LIN {X 0,Y 361.858,Z 207.02,A -85,B 0,C 180,E1 -12997.223,E2 -12997.223} C_VEL
LIN {X 0,Y 361.83,Z 207.034,A -85,B 0,C 180,E1 -13000.756,E2 -13000.756} C_VEL
LIN {X 0,Y 361.812,Z 207.04,A -85,B 0,C 180,E1 -13004.369,E2 -13004.369} C_VEL
LIN {X 0,Y 361.828,Z 207.039,A -85,B 0,C 180,E1 -13007.569,E2 -13007.569} C_VEL
LIN {X 0,Y 361.879,Z 207.126,A -85,B 0,C 180,E1 -13011.447,E2 -13011.447} C_VEL
LIN {X 0,Y 365.809,Z 219.947,A -85,B 0,C 180,E1 -13014.488,E2 -13014.488} C_VEL
LIN {X 0,Y 369.445,Z 233.39,A -85,B 0,C 180,E1 -13017.402,E2 -13017.402} C_VEL
LIN {X 0,Y 372.235,Z 244.85,A -85,B 0,C 180,E1 -13019.72,E2 -13019.72} C_VEL
LIN {X 0,Y 373.066,Z 248.951,A -85,B 0,C 180,E1 -13019.921,E2 -13019.921} C_VEL
LIN {X 0,Y 377.476,Z 275.58,A -85,B 0,C 180,E1 -13020.87,E2 -13020.87} C_VEL
LIN {X 0,Y 378.031,Z 280.109,A -85,B 0,C 180,E1 -13021.013,E2 -13021.013} C_VEL
LIN {X 0,Y 374.715,Z 405.34,A -85,B 0,C 180,E1 -13023.549,E2 -13023.549} C_VEL
LIN {X 0,Y 373.825,Z 420.56,A -85,B 0,C 180,E1 -13024.044,E2 -13024.044} C_VEL
LIN {X 0,Y 372.576,Z 436.071,A -85,B 0,C 180,E1 -13024.78,E2 -13024.78} C_VEL
LIN {X 0,Y 371.215,Z 450.264,A -85,B 0,C 180,E1 -13025.684,E2 -13025.684} C_VEL
LIN {X 0,Y 369.635,Z 463.713,A -85,B 0,C 180,E1 -13026.764,E2 -13026.764} C_VEL
LIN {X 0,Y 367.883,Z 477.375,A -85,B 0,C 180,E1 -13028.129,E2 -13028.129} C_VEL
LIN {X 0,Y 366.23,Z 489.771,A -85,B 0,C 180,E1 -13029.647,E2 -13029.647} C_VEL
LIN {X 0,Y 364.935,Z 500.221,A -85,B 0,C 180,E1 -13031.182,E2 -13031.182} C_VEL
LIN {X 0,Y 363.602,Z 509.844,A -85,B 0,C 180,E1 -13032.857,E2 -13032.857} C_VEL
LIN {X 0,Y 362.442,Z 519.299,A -85,B 0,C 180,E1 -13034.825,E2 -13034.825} C_VEL
LIN {X 0,Y 361.565,Z 527.133,A -85,B 0,C 180,E1 -13036.798,E2 -13036.798} C_VEL
LIN {X 0,Y 360.999,Z 533.592,A -85,B 0,C 180,E1 -13038.774,E2 -13038.774} C_VEL
LIN {X 0,Y 360.557,Z 539.494,A -85,B 0,C 180,E1 -13041.029,E2 -13041.029} C_VEL
LIN {X 0,Y 360.387,Z 543.966,A -85,B 0,C 180,E1 -13043.281,E2 -13043.281} C_VEL
LIN {X 0,Y 360.351,Z 547.107,A -85,B 0,C 180,E1 -13045.526,E2 -13045.526} C_VEL
LIN {X 0,Y 360.384,Z 548.979,A -85,B 0,C 180,E1 -13047.765,E2 -13047.765} C_VEL
LIN {X 0,Y 360.474,Z 549.615,A -85,B 0,C 180,E1 -13050,E2 -13050} C_VEL
LIN {X 0,Y 360.384,Z 548.971,A -85,B 0,C 180,E1 -13052.236,E2 -13052.236} C_VEL
LIN {X 0,Y 360.384,Z 547.091,A -85,B 0,C 180,E1 -13054.474,E2 -13054.474} C_VEL
LIN {X 0,Y 360.477,Z 543.95,A -85,B 0,C 180,E1 -13056.718,E2 -13056.718} C_VEL
LIN {X 0,Y 360.559,Z 539.471,A -85,B 0,C 180,E1 -13058.971,E2 -13058.971} C_VEL
LIN {X 0,Y 361.002,Z 533.555,A -85,B 0,C 180,E1 -13061.226,E2 -13061.226} C_VEL
LIN {X 0,Y 361.685,Z 526.041,A -85,B 0,C 180,E1 -13063.484,E2 -13063.484} C_VEL
LIN {X 0,Y 362.613,Z 517.975,A -85,B 0,C 180,E1 -13065.456,E2 -13065.456} C_VEL
LIN {X 0,Y 363.789,Z 508.252,A -85,B 0,C 180,E1 -13067.424,E2 -13067.424} C_VEL
LIN {X 0,Y 365.118,Z 498.314,A -85,B 0,C 180,E1 -13069.101,E2 -13069.101} C_VEL
LIN {X 0,Y 366.636,Z 486.473,A -85,B 0,C 180,E1 -13070.771,E2 -13070.771} C_VEL
LIN {X 0,Y 368.201,Z 474.69,A -85,B 0,C 180,E1 -13072.147,E2 -13072.147} C_VEL
LIN {X 0,Y 369.832,Z 461.965,A -85,B 0,C 180,E1 -13073.372,E2 -13073.372} C_VEL
LIN {X 0,Y 371.43,Z 448.089,A -85,B 0,C 180,E1 -13074.451,E2 -13074.451} C_VEL
LIN {X 0,Y 372.66,Z 434.821,A -85,B 0,C 180,E1 -13075.275,E2 -13075.275} C_VEL
LIN {X 0,Y 373.81,Z 420.208,A -85,B 0,C 180,E1 -13075.958,E2 -13075.958} C_VEL
LIN {X 0,Y 374.684,Z 404.745,A -85,B 0,C 180,E1 -13076.454,E2 -13076.454} C_VEL
LIN {X 0,Y 377.559,Z 296.462,A -85,B 0,C 180,E1 -13078.649,E2 -13078.649} C_VEL
LIN {X 0,Y 377.872,Z 278.457,A -85,B 0,C 180,E1 -13079.019,E2 -13079.019} C_VEL
LIN {X 0,Y 372.834,Z 247.587,A -85,B 0,C 180,E1 -13080.112,E2 -13080.112} C_VEL
LIN {X 0,Y 372.193,Z 244.833,A -85,B 0,C 180,E1 -13080.272,E2 -13080.272} C_VEL
LIN {X 0,Y 369.443,Z 233.326,A -85,B 0,C 180,E1 -13082.6,E2 -13082.6} C_VEL
LIN {X 0,Y 365.814,Z 219.862,A -85,B 0,C 180,E1 -13085.517,E2 -13085.517} C_VEL
LIN {X 0,Y 361.901,Z 207.157,A -85,B 0,C 180,E1 -13088.533,E2 -13088.533} C_VEL
LIN {X 0,Y 361.82,Z 207.013,A -85,B 0,C 180,E1 -13091.331,E2 -13091.331} C_VEL
LIN {X 0,Y 361.815,Z 207.03,A -85,B 0,C 180,E1 -13094.369,E2 -13094.369} C_VEL
LIN {X 0,Y 361.834,Z 207.026,A -85,B 0,C 180,E1 -13097.568,E2 -13097.568} C_VEL
LIN {X 0,Y 361.868,Z 207.03,A -85,B 0,C 180,E1 -13100.973,E2 -13100.973} C_VEL
LIN {X 0,Y 361.872,Z 207.038,A -85,B 0,C 180,E1 -13104.655,E2 -13104.655} C_VEL
LIN {X 0,Y 361.835,Z 207.02,A -85,B 0,C 180,E1 -13108.371,E2 -13108.371} C_VEL
LIN {X 0,Y 361.899,Z 207.028,A -85,B 0,C 180,E1 -13110.955,E2 -13110.955} C_VEL
LIN {X 0,Y 361.952,Z 206.995,A -85,B 0,C 180,E1 -13113.475,E2 -13113.475} C_VEL
LIN {X 0,Y 361.888,Z 207.03,A -85,B 0,C 180,E1 -13117.145,E2 -13117.145} C_VEL
LIN {X 0,Y 361.919,Z 207.026,A -85,B 0,C 180,E1 -13120.724,E2 -13120.724} C_VEL
LIN {X 0,Y 361.944,Z 207.026,A -85,B 0,C 180,E1 -13124.226,E2 -13124.226} C_VEL
LIN {X 0,Y 361.997,Z 207.012,A -85,B 0,C 180,E1 -13126.528,E2 -13126.528} C_VEL
LIN {X 0,Y 362.029,Z 207.007,A -85,B 0,C 180,E1 -13129.938,E2 -13129.938} C_VEL
LIN {X 0,Y 362.161,Z 206.997,A -85,B 0,C 180,E1 -13133.314,E2 -13133.314} C_VEL
LIN {X 0,Y 362.278,Z 206.978,A -85,B 0,C 180,E1 -13137.777,E2 -13137.777} C_VEL
LIN {X 0,Y 362.424,Z 206.963,A -85,B 0,C 180,E1 -13140,E2 -13140} C_VEL
LIN {X 0,Y 362.278,Z 206.977,A -85,B 0,C 180,E1 -13142.224,E2 -13142.224} C_VEL
LIN {X 0,Y 362.17,Z 206.993,A -85,B 0,C 180,E1 -13146.686,E2 -13146.686} C_VEL
LIN {X 0,Y 362.073,Z 207.005,A -85,B 0,C 180,E1 -13148.933,E2 -13148.933} C_VEL
LIN {X 0,Y 361.958,Z 207.015,A -85,B 0,C 180,E1 -13152.333,E2 -13152.333} C_VEL
LIN {X 0,Y 361.961,Z 207.022,A -85,B 0,C 180,E1 -13154.621,E2 -13154.621} C_VEL
LIN {X 0,Y 361.955,Z 207.022,A -85,B 0,C 180,E1 -13158.1,E2 -13158.1} C_VEL
LIN {X 0,Y 361.892,Z 207.031,A -85,B 0,C 180,E1 -13161.653,E2 -13161.653} C_VEL
LIN {X 0,Y 361.927,Z 207.029,A -85,B 0,C 180,E1 -13165.29,E2 -13165.29} C_VEL
LIN {X 0,Y 361.907,Z 207.01,A -85,B 0,C 180,E1 -13167.779,E2 -13167.779} C_VEL
LIN {X 0,Y 361.837,Z 207.038,A -85,B 0,C 180,E1 -13171.63,E2 -13171.63} C_VEL
LIN {X 0,Y 361.874,Z 207.015,A -85,B 0,C 180,E1 -13175.345,E2 -13175.345} C_VEL
LIN {X 0,Y 361.869,Z 207.02,A -85,B 0,C 180,E1 -13179.027,E2 -13179.027} C_VEL
LIN {X 0,Y 361.836,Z 207.035,A -85,B 0,C 180,E1 -13182.829,E2 -13182.829} C_VEL
LIN {X 0,Y 361.819,Z 207.041,A -85,B 0,C 180,E1 -13185.947,E2 -13185.947} C_VEL
LIN {X 0,Y 361.837,Z 207.04,A -85,B 0,C 180,E1 -13189.245,E2 -13189.245} C_VEL
LIN {X 0,Y 361.872,Z 207.03,A -85,B 0,C 180,E1 -13192.776,E2 -13192.776} C_VEL
LIN {X 0,Y 361.897,Z 207.231,A -85,B 0,C 180,E1 -13193.593,E2 -13193.593} C_VEL
LIN {X 0,Y 364.857,Z 217.605,A -85,B 0,C 180,E1 -13196.315,E2 -13196.315} C_VEL
LIN {X 0,Y 367.533,Z 228.193,A -85,B 0,C 180,E1 -13198.916,E2 -13198.916} C_VEL
LIN {X 0,Y 370.249,Z 240.049,A -85,B 0,C 180,E1 -13201.67,E2 -13201.67} C_VEL
LIN {X 0,Y 370.322,Z 243.02,A -85,B 0,C 180,E1 -13202.292,E2 -13202.292} C_VEL
LIN {X 0,Y 370.224,Z 244.579,A -85,B 0,C 180,E1 -13202.552,E2 -13202.552} C_VEL
LIN {X 0,Y 376.066,Z 272.726,A -85,B 0,C 180,E1 -13203.636,E2 -13203.636} C_VEL
LIN {X 0,Y 377.412,Z 280.727,A -85,B 0,C 180,E1 -13203.904,E2 -13203.904} C_VEL
LIN {X 0,Y 375.224,Z 388.776,A -85,B 0,C 180,E1 -13205.886,E2 -13205.886} C_VEL
LIN {X 0,Y 374.523,Z 402.901,A -85,B 0,C 180,E1 -13206.353,E2 -13206.353} C_VEL
LIN {X 0,Y 373.655,Z 416.248,A -85,B 0,C 180,E1 -13207.005,E2 -13207.005} C_VEL
LIN {X 0,Y 372.396,Z 429.002,A -85,B 0,C 180,E1 -13207.824,E2 -13207.824} C_VEL
LIN {X 0,Y 371.049,Z 441.949,A -85,B 0,C 180,E1 -13208.907,E2 -13208.907} C_VEL
LIN {X 0,Y 369.441,Z 453.698,A -85,B 0,C 180,E1 -13210.12,E2 -13210.12} C_VEL
LIN {X 0,Y 368.1,Z 463.475,A -85,B 0,C 180,E1 -13211.349,E2 -13211.349} C_VEL
LIN {X 0,Y 366.399,Z 474.26,A -85,B 0,C 180,E1 -13212.991,E2 -13212.991} C_VEL
LIN {X 0,Y 365.128,Z 483.181,A -85,B 0,C 180,E1 -13214.653,E2 -13214.653} C_VEL
LIN {X 0,Y 363.659,Z 491.735,A -85,B 0,C 180,E1 -13216.59,E2 -13216.59} C_VEL
LIN {X 0,Y 362.727,Z 497.801,A -85,B 0,C 180,E1 -13218.261,E2 -13218.261} C_VEL
LIN {X 0,Y 361.781,Z 504.251,A -85,B 0,C 180,E1 -13220.495,E2 -13220.495} C_VEL
LIN {X 0,Y 361.304,Z 508.07,A -85,B 0,C 180,E1 -13222.174,E2 -13222.174} C_VEL
LIN {X 0,Y 360.869,Z 511.89,A -85,B 0,C 180,E1 -13224.412,E2 -13224.412} C_VEL
LIN {X 0,Y 360.604,Z 514.38,A -85,B 0,C 180,E1 -13226.648,E2 -13226.648} C_VEL
LIN {X 0,Y 360.499,Z 515.621,A -85,B 0,C 180,E1 -13228.883,E2 -13228.883} C_VEL
LIN {X 0,Y 360.497,Z 515.649,A -85,B 0,C 180,E1 -13231.117,E2 -13231.117} C_VEL
LIN {X 0,Y 360.594,Z 514.467,A -85,B 0,C 180,E1 -13233.352,E2 -13233.352} C_VEL
LIN {X 0,Y 360.857,Z 512.038,A -85,B 0,C 180,E1 -13235.588,E2 -13235.588} C_VEL
LIN {X 0,Y 361.286,Z 508.284,A -85,B 0,C 180,E1 -13237.826,E2 -13237.826} C_VEL
LIN {X 0,Y 361.943,Z 503.077,A -85,B 0,C 180,E1 -13240.064,E2 -13240.064} C_VEL
LIN {X 0,Y 362.965,Z 496.242,A -85,B 0,C 180,E1 -13242.297,E2 -13242.297} C_VEL
LIN {X 0,Y 364.222,Z 488.716,A -85,B 0,C 180,E1 -13244.242,E2 -13244.242} C_VEL
LIN {X 0,Y 365.555,Z 479.746,A -85,B 0,C 180,E1 -13246.129,E2 -13246.129} C_VEL
LIN {X 0,Y 366.277,Z 475.133,A -85,B 0,C 180,E1 -13246.961,E2 -13246.961} C_VEL
LIN {X 0,Y 366.252,Z 471.21,A -85,B 0,C 180,E1 -13247.651,E2 -13247.651} C_VEL
LIN {X 0,Y 364.53,Z 464.68,A -85,B 0,C 180,E1 -13248.791,E2 -13248.791} C_VEL
LIN {X 0,Y 362.904,Z 457.796,A -85,B 0,C 180,E1 -13249.881,E2 -13249.881} C_VEL
LIN {X 0,Y 362.989,Z 453.195,A -85,B 0,C 180,E1 -13250.469,E2 -13250.469} C_VEL
LIN {X 0,Y 364.736,Z 440.566,A -85,B 0,C 180,E1 -13251.772,E2 -13251.772} C_VEL
LIN {X 0,Y 366.108,Z 427.91,A -85,B 0,C 180,E1 -13252.814,E2 -13252.814} C_VEL
LIN {X 0,Y 367.367,Z 414.082,A -85,B 0,C 180,E1 -13253.687,E2 -13253.687} C_VEL
LIN {X 0,Y 368.307,Z 400.048,A -85,B 0,C 180,E1 -13254.333,E2 -13254.333} C_VEL
LIN {X 0,Y 368.949,Z 385.269,A -85,B 0,C 180,E1 -13254.775,E2 -13254.775} C_VEL
LIN {X 0,Y 371.083,Z 280.253,A -85,B 0,C 180,E1 -13256.723,E2 -13256.723} C_VEL
LIN {X 0,Y 364.68,Z 248.87,A -85,B 0,C 180,E1 -13257.924,E2 -13257.924} C_VEL
LIN {X 0,Y 363.707,Z 244.456,A -85,B 0,C 180,E1 -13258.139,E2 -13258.139} C_VEL
LIN {X 0,Y 363.246,Z 240.748,A -85,B 0,C 180,E1 -13258.926,E2 -13258.926} C_VEL
LIN {X 0,Y 360.536,Z 228.921,A -85,B 0,C 180,E1 -13261.756,E2 -13261.756} C_VEL
LIN {X 0,Y 357.479,Z 217.065,A -85,B 0,C 180,E1 -13264.759,E2 -13264.759} C_VEL
LIN {X 0,Y 354.825,Z 207.985,A -85,B 0,C 180,E1 -13267.271,E2 -13267.271} C_VEL
LIN {X 0,Y 354.786,Z 207.92,A -85,B 0,C 180,E1 -13270.82,E2 -13270.82} C_VEL
LIN {X 0,Y 354.761,Z 207.919,A -85,B 0,C 180,E1 -13274.506,E2 -13274.506} C_VEL
LIN {X 0,Y 354.791,Z 207.918,A -85,B 0,C 180,E1 -13277.662,E2 -13277.662} C_VEL
LIN {X 0,Y 354.811,Z 207.897,A -85,B 0,C 180,E1 -13280.665,E2 -13280.665} C_VEL
LIN {X 0,Y 354.818,Z 207.899,A -85,B 0,C 180,E1 -13284.3,E2 -13284.3} C_VEL
LIN {X 0,Y 354.785,Z 207.918,A -85,B 0,C 180,E1 -13287.666,E2 -13287.666} C_VEL
LIN {X 0,Y 354.864,Z 207.882,A -85,B 0,C 180,E1 -13290.621,E2 -13290.621} C_VEL
LIN {X 0,Y 354.894,Z 207.901,A -85,B 0,C 180,E1 -13294.172,E2 -13294.172} C_VEL
LIN {X 0,Y 354.829,Z 207.91,A -85,B 0,C 180,E1 -13297.893,E2 -13297.893} C_VEL
LIN {X 0,Y 354.917,Z 207.899,A -85,B 0,C 180,E1 -13301.891,E2 -13301.891} C_VEL
LIN {X 0,Y 354.936,Z 207.897,A -85,B 0,C 180,E1 -13305.981,E2 -13305.981} C_VEL
LIN {X 0,Y 354.971,Z 207.891,A -85,B 0,C 180,E1 -13309.735,E2 -13309.735} C_VEL
LIN {X 0,Y 355.107,Z 207.869,A -85,B 0,C 180,E1 -13312.037,E2 -13312.037} C_VEL
LIN {X 0,Y 355.086,Z 207.879,A -85,B 0,C 180,E1 -13314.32,E2 -13314.32} C_VEL
LIN {X 0,Y 355.239,Z 207.853,A -85,B 0,C 180,E1 -13317.732,E2 -13317.732} C_VEL
LIN {X 0,Y 355.391,Z 207.839,A -85,B 0,C 180,E1 -13320,E2 -13320} C_VEL
LIN {X 0,Y 355.239,Z 207.854,A -85,B 0,C 180,E1 -13322.267,E2 -13322.267} C_VEL
LIN {X 0,Y 355.131,Z 207.873,A -85,B 0,C 180,E1 -13326.819,E2 -13326.819} C_VEL
LIN {X 0,Y 355.008,Z 207.882,A -85,B 0,C 180,E1 -13329.112,E2 -13329.112} C_VEL
LIN {X 0,Y 354.914,Z 207.897,A -85,B 0,C 180,E1 -13332.581,E2 -13332.581} C_VEL
LIN {X 0,Y 354.883,Z 207.905,A -85,B 0,C 180,E1 -13336.096,E2 -13336.096} C_VEL
LIN {X 0,Y 354.9,Z 207.898,A -85,B 0,C 180,E1 -13338.472,E2 -13338.472} C_VEL
LIN {X 0,Y 354.828,Z 207.907,A -85,B 0,C 180,E1 -13342.106,E2 -13342.106} C_VEL
LIN {X 0,Y 354.893,Z 207.877,A -85,B 0,C 180,E1 -13345.828,E2 -13345.828} C_VEL
LIN {X 0,Y 354.848,Z 207.912,A -85,B 0,C 180,E1 -13349.679,E2 -13349.679} C_VEL
LIN {X 0,Y 354.8,Z 207.899,A -85,B 0,C 180,E1 -13353.702,E2 -13353.702} C_VEL
LIN {X 0,Y 354.792,Z 207.907,A -85,B 0,C 180,E1 -13356.46,E2 -13356.46} C_VEL
LIN {X 0,Y 354.819,Z 207.912,A -85,B 0,C 180,E1 -13359.424,E2 -13359.424} C_VEL
LIN {X 0,Y 354.783,Z 207.908,A -85,B 0,C 180,E1 -13362.868,E2 -13362.868} C_VEL
LIN {X 0,Y 354.761,Z 207.91,A -85,B 0,C 180,E1 -13366.104,E2 -13366.104} C_VEL
LIN {X 0,Y 354.777,Z 207.88,A -85,B 0,C 180,E1 -13369.179,E2 -13369.179} C_VEL
LIN {X 0,Y 354.846,Z 208.08,A -85,B 0,C 180,E1 -13370.784,E2 -13370.784} C_VEL
LIN {X 0,Y 358.939,Z 221.433,A -85,B 0,C 180,E1 -13374.029,E2 -13374.029} C_VEL
LIN {X 0,Y 362.471,Z 234.285,A -85,B 0,C 180,E1 -13376.904,E2 -13376.904} C_VEL
LIN {X 0,Y 365.188,Z 245.142,A -85,B 0,C 180,E1 -13379.137,E2 -13379.137} C_VEL
LIN {X 0,Y 366.628,Z 248.786,A -85,B 0,C 180,E1 -13379.367,E2 -13379.367} C_VEL
LIN {X 0,Y 370.877,Z 274.547,A -85,B 0,C 180,E1 -13380.311,E2 -13380.311} C_VEL
LIN {X 0,Y 371.729,Z 281.26,A -85,B 0,C 180,E1 -13380.531,E2 -13380.531} C_VEL
LIN {X 0,Y 368.294,Z 405.657,A -85,B 0,C 180,E1 -13383.089,E2 -13383.089} C_VEL
LIN {X 0,Y 367.319,Z 421.492,A -85,B 0,C 180,E1 -13383.626,E2 -13383.626} C_VEL
LIN {X 0,Y 366.057,Z 436.211,A -85,B 0,C 180,E1 -13384.345,E2 -13384.345} C_VEL
LIN {X 0,Y 364.716,Z 449.758,A -85,B 0,C 180,E1 -13385.222,E2 -13385.222} C_VEL
LIN {X 0,Y 363.065,Z 463.252,A -85,B 0,C 180,E1 -13386.318,E2 -13386.318} C_VEL
LIN {X 0,Y 361.254,Z 476.962,A -85,B 0,C 180,E1 -13387.707,E2 -13387.707} C_VEL
LIN {X 0,Y 359.509,Z 489.38,A -85,B 0,C 180,E1 -13389.249,E2 -13389.249} C_VEL
LIN {X 0,Y 358.111,Z 499.836,A -85,B 0,C 180,E1 -13390.81,E2 -13390.81} C_VEL
LIN {X 0,Y 356.744,Z 509.473,A -85,B 0,C 180,E1 -13392.517,E2 -13392.517} C_VEL
LIN {X 0,Y 355.511,Z 518.939,A -85,B 0,C 180,E1 -13394.522,E2 -13394.522} C_VEL
LIN {X 0,Y 354.555,Z 526.779,A -85,B 0,C 180,E1 -13396.532,E2 -13396.532} C_VEL
LIN {X 0,Y 353.952,Z 533.245,A -85,B 0,C 180,E1 -13398.548,E2 -13398.548} C_VEL
LIN {X 0,Y 353.498,Z 539.153,A -85,B 0,C 180,E1 -13400.849,E2 -13400.849} C_VEL
LIN {X 0,Y 353.305,Z 543.629,A -85,B 0,C 180,E1 -13403.146,E2 -13403.146} C_VEL
LIN {X 0,Y 353.262,Z 546.772,A -85,B 0,C 180,E1 -13405.436,E2 -13405.436} C_VEL
LIN {X 0,Y 353.285,Z 548.646,A -85,B 0,C 180,E1 -13407.72,E2 -13407.72} C_VEL
LIN {X 0,Y 353.393,Z 549.283,A -85,B 0,C 180,E1 -13410,E2 -13410} C_VEL
LIN {X 0,Y 353.285,Z 548.638,A -85,B 0,C 180,E1 -13412.281,E2 -13412.281} C_VEL
LIN {X 0,Y 353.295,Z 546.756,A -85,B 0,C 180,E1 -13414.564,E2 -13414.564} C_VEL
LIN {X 0,Y 353.383,Z 543.611,A -85,B 0,C 180,E1 -13416.854,E2 -13416.854} C_VEL
LIN {X 0,Y 353.499,Z 539.128,A -85,B 0,C 180,E1 -13419.152,E2 -13419.152} C_VEL
LIN {X 0,Y 353.957,Z 533.206,A -85,B 0,C 180,E1 -13421.453,E2 -13421.453} C_VEL
LIN {X 0,Y 354.72,Z 525.687,A -85,B 0,C 180,E1 -13423.754,E2 -13423.754} C_VEL
LIN {X 0,Y 355.674,Z 517.61,A -85,B 0,C 180,E1 -13425.765,E2 -13425.765} C_VEL
LIN {X 0,Y 356.957,Z 507.879,A -85,B 0,C 180,E1 -13427.769,E2 -13427.769} C_VEL
LIN {X 0,Y 358.534,Z 496.723,A -85,B 0,C 180,E1 -13429.663,E2 -13429.663} C_VEL
LIN {X 0,Y 359.929,Z 486.064,A -85,B 0,C 180,E1 -13431.176,E2 -13431.176} C_VEL
LIN {X 0,Y 361.605,Z 474.256,A -85,B 0,C 180,E1 -13432.573,E2 -13432.573} C_VEL
LIN {X 0,Y 363.245,Z 461.488,A -85,B 0,C 180,E1 -13433.821,E2 -13433.821} C_VEL
LIN {X 0,Y 364.918,Z 447.555,A -85,B 0,C 180,E1 -13434.916,E2 -13434.916} C_VEL
LIN {X 0,Y 366.277,Z 433.522,A -85,B 0,C 180,E1 -13435.787,E2 -13435.787} C_VEL
LIN {X 0,Y 367.489,Z 418.521,A -85,B 0,C 180,E1 -13436.477,E2 -13436.477} C_VEL
LIN {X 0,Y 368.325,Z 403.593,A -85,B 0,C 180,E1 -13436.947,E2 -13436.947} C_VEL
LIN {X 0,Y 371.686,Z 280.699,A -85,B 0,C 180,E1 -13439.467,E2 -13439.467} C_VEL
LIN {X 0,Y 367.099,Z 251.451,A -85,B 0,C 180,E1 -13440.514,E2 -13440.514} C_VEL
LIN {X 0,Y 366.131,Z 247.57,A -85,B 0,C 180,E1 -13440.687,E2 -13440.687} C_VEL
LIN {X 0,Y 365.05,Z 244.821,A -85,B 0,C 180,E1 -13440.891,E2 -13440.891} C_VEL
LIN {X 0,Y 362.081,Z 232.745,A -85,B 0,C 180,E1 -13443.423,E2 -13443.423} C_VEL
LIN {X 0,Y 358.606,Z 220.27,A -85,B 0,C 180,E1 -13446.224,E2 -13446.224} C_VEL
LIN {X 0,Y 354.843,Z 208.045,A -85,B 0,C 180,E1 -13449.217,E2 -13449.217} C_VEL
LIN {X 0,Y 354.785,Z 207.919,A -85,B 0,C 180,E1 -13452.867,E2 -13452.867} C_VEL
LIN {X 0,Y 354.766,Z 207.92,A -85,B 0,C 180,E1 -13456.104,E2 -13456.104} C_VEL
LIN {X 0,Y 354.786,Z 207.911,A -85,B 0,C 180,E1 -13459.179,E2 -13459.179} C_VEL
LIN {X 0,Y 354.806,Z 207.898,A -85,B 0,C 180,E1 -13462.403,E2 -13462.403} C_VEL
LIN {X 0,Y 354.81,Z 207.916,A -85,B 0,C 180,E1 -13464.941,E2 -13464.941} C_VEL
LIN {X 0,Y 354.791,Z 207.897,A -85,B 0,C 180,E1 -13468.405,E2 -13468.405} C_VEL
LIN {X 0,Y 354.849,Z 207.9,A -85,B 0,C 180,E1 -13471.619,E2 -13471.619} C_VEL
LIN {X 0,Y 354.897,Z 207.876,A -85,B 0,C 180,E1 -13474.173,E2 -13474.173} C_VEL
LIN {X 0,Y 354.833,Z 207.907,A -85,B 0,C 180,E1 -13477.894,E2 -13477.894} C_VEL
LIN {X 0,Y 354.921,Z 207.894,A -85,B 0,C 180,E1 -13481.891,E2 -13481.891} C_VEL
LIN {X 0,Y 354.941,Z 207.89,A -85,B 0,C 180,E1 -13485.981,E2 -13485.981} C_VEL
LIN {X 0,Y 354.976,Z 207.886,A -85,B 0,C 180,E1 -13489.736,E2 -13489.736} C_VEL
LIN {X 0,Y 355.124,Z 207.873,A -85,B 0,C 180,E1 -13493.181,E2 -13493.181} C_VEL
LIN {X 0,Y 355.242,Z 207.855,A -85,B 0,C 180,E1 -13497.733,E2 -13497.733} C_VEL
LIN {X 0,Y 355.373,Z 207.841,A -85,B 0,C 180,E1 -13500,E2 -13500} C_VEL
LIN {X 0,Y 355.242,Z 207.853,A -85,B 0,C 180,E1 -13502.268,E2 -13502.268} C_VEL
LIN {X 0,Y 355.136,Z 207.868,A -85,B 0,C 180,E1 -13506.819,E2 -13506.819} C_VEL
LIN {X 0,Y 355.014,Z 207.886,A -85,B 0,C 180,E1 -13509.113,E2 -13509.113} C_VEL
LIN {X 0,Y 354.919,Z 207.892,A -85,B 0,C 180,E1 -13512.581,E2 -13512.581} C_VEL
LIN {X 0,Y 354.888,Z 207.894,A -85,B 0,C 180,E1 -13516.096,E2 -13516.096} C_VEL
LIN {X 0,Y 354.9,Z 207.901,A -85,B 0,C 180,E1 -13518.472,E2 -13518.472} C_VEL
LIN {X 0,Y 354.835,Z 207.909,A -85,B 0,C 180,E1 -13522.106,E2 -13522.106} C_VEL
LIN {X 0,Y 354.898,Z 207.901,A -85,B 0,C 180,E1 -13525.828,E2 -13525.828} C_VEL
LIN {X 0,Y 354.817,Z 207.891,A -85,B 0,C 180,E1 -13529.682,E2 -13529.682} C_VEL
LIN {X 0,Y 354.814,Z 207.899,A -85,B 0,C 180,E1 -13533.684,E2 -13533.684} C_VEL
LIN {X 0,Y 354.798,Z 207.908,A -85,B 0,C 180,E1 -13536.46,E2 -13536.46} C_VEL
LIN {X 0,Y 354.824,Z 207.894,A -85,B 0,C 180,E1 -13539.424,E2 -13539.424} C_VEL
LIN {X 0,Y 354.788,Z 207.912,A -85,B 0,C 180,E1 -13542.867,E2 -13542.867} C_VEL
LIN {X 0,Y 354.768,Z 207.92,A -85,B 0,C 180,E1 -13546.104,E2 -13546.104} C_VEL
LIN {X 0,Y 354.789,Z 207.918,A -85,B 0,C 180,E1 -13549.179,E2 -13549.179} C_VEL
LIN {X 0,Y 354.849,Z 208.012,A -85,B 0,C 180,E1 -13552.883,E2 -13552.883} C_VEL
LIN {X 0,Y 358.303,Z 220.102,A -85,B 0,C 180,E1 -13556.152,E2 -13556.152} C_VEL
LIN {X 0,Y 361.062,Z 231.207,A -85,B 0,C 180,E1 -13558.921,E2 -13558.921} C_VEL
LIN {X 0,Y 363.456,Z 241.708,A -85,B 0,C 180,E1 -13561.407,E2 -13561.407} C_VEL
LIN {X 0,Y 363.677,Z 244.442,A -85,B 0,C 180,E1 -13561.966,E2 -13561.966} C_VEL
LIN {X 0,Y 369.097,Z 270.076,A -85,B 0,C 180,E1 -13563.008,E2 -13563.008} C_VEL
LIN {X 0,Y 371.088,Z 280.716,A -85,B 0,C 180,E1 -13563.393,E2 -13563.393} C_VEL
LIN {X 0,Y 368.853,Z 388.562,A -85,B 0,C 180,E1 -13565.405,E2 -13565.405} C_VEL
LIN {X 0,Y 368.114,Z 402.833,A -85,B 0,C 180,E1 -13565.878,E2 -13565.878} C_VEL
LIN {X 0,Y 367.147,Z 416.969,A -85,B 0,C 180,E1 -13566.583,E2 -13566.583} C_VEL
LIN {X 0,Y 365.866,Z 429.497,A -85,B 0,C 180,E1 -13567.407,E2 -13567.407} C_VEL
LIN {X 0,Y 364.447,Z 442.397,A -85,B 0,C 180,E1 -13568.506,E2 -13568.506} C_VEL
LIN {X 0,Y 362.78,Z 454.113,A -85,B 0,C 180,E1 -13569.74,E2 -13569.74} C_VEL
LIN {X 0,Y 361.378,Z 463.866,A -85,B 0,C 180,E1 -13570.989,E2 -13570.989} C_VEL
LIN {X 0,Y 359.604,Z 474.634,A -85,B 0,C 180,E1 -13572.66,E2 -13572.66} C_VEL
LIN {X 0,Y 358.266,Z 483.544,A -85,B 0,C 180,E1 -13574.352,E2 -13574.352} C_VEL
LIN {X 0,Y 356.764,Z 492.088,A -85,B 0,C 180,E1 -13576.326,E2 -13576.326} C_VEL
LIN {X 0,Y 355.775,Z 498.146,A -85,B 0,C 180,E1 -13578.029,E2 -13578.029} C_VEL
LIN {X 0,Y 354.784,Z 504.591,A -85,B 0,C 180,E1 -13580.306,E2 -13580.306} C_VEL
LIN {X 0,Y 354.264,Z 508.41,A -85,B 0,C 180,E1 -13582.017,E2 -13582.017} C_VEL
LIN {X 0,Y 353.825,Z 512.225,A -85,B 0,C 180,E1 -13584.3,E2 -13584.3} C_VEL
LIN {X 0,Y 353.516,Z 514.715,A -85,B 0,C 180,E1 -13586.58,E2 -13586.58} C_VEL
LIN {X 0,Y 353.421,Z 515.954,A -85,B 0,C 180,E1 -13588.86,E2 -13588.86} C_VEL
LIN {X 0,Y 353.418,Z 515.981,A -85,B 0,C 180,E1 -13591.139,E2 -13591.139} C_VEL
LIN {X 0,Y 353.505,Z 514.8,A -85,B 0,C 180,E1 -13593.419,E2 -13593.419} C_VEL
LIN {X 0,Y 353.792,Z 512.372,A -85,B 0,C 180,E1 -13595.7,E2 -13595.7} C_VEL
LIN {X 0,Y 354.241,Z 508.621,A -85,B 0,C 180,E1 -13597.982,E2 -13597.982} C_VEL
LIN {X 0,Y 354.94,Z 503.419,A -85,B 0,C 180,E1 -13600.265,E2 -13600.265} C_VEL
LIN {X 0,Y 356.011,Z 496.588,A -85,B 0,C 180,E1 -13602.541,E2 -13602.541} C_VEL
LIN {X 0,Y 357.333,Z 489.07,A -85,B 0,C 180,E1 -13604.522,E2 -13604.522} C_VEL
LIN {X 0,Y 358.738,Z 480.108,A -85,B 0,C 180,E1 -13606.444,E2 -13606.444} C_VEL
LIN {X 0,Y 360.4,Z 470.14,A -85,B 0,C 180,E1 -13608.18,E2 -13608.18} C_VEL
LIN {X 0,Y 362.052,Z 459.413,A -85,B 0,C 180,E1 -13609.71,E2 -13609.71} C_VEL
LIN {X 0,Y 362.989,Z 453.195,A -85,B 0,C 180,E1 -13610.469,E2 -13610.469} C_VEL
LIN {X 0,Y 363.085,Z 448.516,A -85,B 0,C 180,E1 -13611.04,E2 -13611.04} C_VEL
LIN {X 0,Y 361.455,Z 440.814,A -85,B 0,C 180,E1 -13611.999,E2 -13611.999} C_VEL
LIN {X 0,Y 359.744,Z 432.759,A -85,B 0,C 180,E1 -13612.877,E2 -13612.877} C_VEL
LIN {X 0,Y 359.693,Z 427.53,A -85,B 0,C 180,E1 -13613.313,E2 -13613.313} C_VEL
LIN {X 0,Y 360.913,Z 414.689,A -85,B 0,C 180,E1 -13614.137,E2 -13614.137} C_VEL
LIN {X 0,Y 361.898,Z 400.827,A -85,B 0,C 180,E1 -13614.793,E2 -13614.793} C_VEL
LIN {X 0,Y 362.568,Z 386.46,A -85,B 0,C 180,E1 -13615.241,E2 -13615.241} C_VEL
LIN {X 0,Y 364.801,Z 281.372,A -85,B 0,C 180,E1 -13617.228,E2 -13617.228} C_VEL
LIN {X 0,Y 359.474,Z 254.909,A -85,B 0,C 180,E1 -13618.261,E2 -13618.261} C_VEL
LIN {X 0,Y 357.173,Z 245.429,A -85,B 0,C 180,E1 -13618.685,E2 -13618.685} C_VEL
LIN {X 0,Y 356.807,Z 244.075,A -85,B 0,C 180,E1 -13618.828,E2 -13618.828} C_VEL
LIN {X 0,Y 354.349,Z 233.053,A -85,B 0,C 180,E1 -13621.477,E2 -13621.477} C_VEL
LIN {X 0,Y 351.349,Z 221.277,A -85,B 0,C 180,E1 -13624.498,E2 -13624.498} C_VEL
LIN {X 0,Y 348.513,Z 211.254,A -85,B 0,C 180,E1 -13627.225,E2 -13627.225} C_VEL
LIN {X 0,Y 347.772,Z 208.86,A -85,B 0,C 180,E1 -13627.988,E2 -13627.988} C_VEL
LIN {X 0,Y 347.748,Z 208.783,A -85,B 0,C 180,E1 -13631.829,E2 -13631.829} C_VEL
LIN {X 0,Y 347.703,Z 208.79,A -85,B 0,C 180,E1 -13635.026,E2 -13635.026} C_VEL
LIN {X 0,Y 347.747,Z 208.795,A -85,B 0,C 180,E1 -13638.396,E2 -13638.396} C_VEL
LIN {X 0,Y 347.77,Z 208.792,A -85,B 0,C 180,E1 -13642.011,E2 -13642.011} C_VEL
LIN {X 0,Y 347.74,Z 208.773,A -85,B 0,C 180,E1 -13645.535,E2 -13645.535} C_VEL
LIN {X 0,Y 347.76,Z 208.781,A -85,B 0,C 180,E1 -13649.653,E2 -13649.653} C_VEL
LIN {X 0,Y 347.847,Z 208.764,A -85,B 0,C 180,E1 -13652.744,E2 -13652.744} C_VEL
LIN {X 0,Y 347.783,Z 208.782,A -85,B 0,C 180,E1 -13656.161,E2 -13656.161} C_VEL
LIN {X 0,Y 347.811,Z 208.776,A -85,B 0,C 180,E1 -13659.909,E2 -13659.909} C_VEL
LIN {X 0,Y 347.86,Z 208.779,A -85,B 0,C 180,E1 -13662.359,E2 -13662.359} C_VEL
LIN {X 0,Y 347.891,Z 208.774,A -85,B 0,C 180,E1 -13665.97,E2 -13665.97} C_VEL
LIN {X 0,Y 347.922,Z 208.769,A -85,B 0,C 180,E1 -13669.525,E2 -13669.525} C_VEL
LIN {X 0,Y 348.067,Z 208.747,A -85,B 0,C 180,E1 -13671.874,E2 -13671.874} C_VEL
LIN {X 0,Y 348.061,Z 208.753,A -85,B 0,C 180,E1 -13674.205,E2 -13674.205} C_VEL
LIN {X 0,Y 348.201,Z 208.73,A -85,B 0,C 180,E1 -13677.686,E2 -13677.686} C_VEL
LIN {X 0,Y 348.339,Z 208.717,A -85,B 0,C 180,E1 -13680,E2 -13680} C_VEL
LIN {X 0,Y 348.202,Z 208.731,A -85,B 0,C 180,E1 -13682.313,E2 -13682.313} C_VEL
LIN {X 0,Y 348.099,Z 208.748,A -85,B 0,C 180,E1 -13686.958,E2 -13686.958} C_VEL
LIN {X 0,Y 347.961,Z 208.76,A -85,B 0,C 180,E1 -13689.298,E2 -13689.298} C_VEL
LIN {X 0,Y 347.883,Z 208.771,A -85,B 0,C 180,E1 -13692.839,E2 -13692.839} C_VEL
LIN {X 0,Y 347.832,Z 208.78,A -85,B 0,C 180,E1 -13696.431,E2 -13696.431} C_VEL
LIN {X 0,Y 347.849,Z 208.778,A -85,B 0,C 180,E1 -13698.86,E2 -13698.86} C_VEL
LIN {X 0,Y 347.768,Z 208.79,A -85,B 0,C 180,E1 -13702.58,E2 -13702.58} C_VEL
LIN {X 0,Y 347.806,Z 208.769,A -85,B 0,C 180,E1 -13705.109,E2 -13705.109} C_VEL
LIN {X 0,Y 347.804,Z 208.765,A -85,B 0,C 180,E1 -13707.694,E2 -13707.694} C_VEL
LIN {X 0,Y 347.758,Z 208.789,A -85,B 0,C 180,E1 -13710.347,E2 -13710.347} C_VEL
LIN {X 0,Y 347.738,Z 208.793,A -85,B 0,C 180,E1 -13714.464,E2 -13714.464} C_VEL
LIN {X 0,Y 347.768,Z 208.774,A -85,B 0,C 180,E1 -13717.989,E2 -13717.989} C_VEL
LIN {X 0,Y 347.745,Z 208.779,A -85,B 0,C 180,E1 -13721.831,E2 -13721.831} C_VEL
LIN {X 0,Y 347.7,Z 208.789,A -85,B 0,C 180,E1 -13725.027,E2 -13725.027} C_VEL
LIN {X 0,Y 347.742,Z 208.769,A -85,B 0,C 180,E1 -13728.398,E2 -13728.398} C_VEL
LIN {X 0,Y 347.771,Z 208.994,A -85,B 0,C 180,E1 -13730.061,E2 -13730.061} C_VEL
LIN {X 0,Y 351.64,Z 221.205,A -85,B 0,C 180,E1 -13733.161,E2 -13733.161} C_VEL
LIN {X 0,Y 355.59,Z 235.255,A -85,B 0,C 180,E1 -13736.4,E2 -13736.4} C_VEL
LIN {X 0,Y 358.055,Z 245.198,A -85,B 0,C 180,E1 -13738.495,E2 -13738.495} C_VEL
LIN {X 0,Y 360.684,Z 251.591,A -85,B 0,C 180,E1 -13738.903,E2 -13738.903} C_VEL
LIN {X 0,Y 364.68,Z 275.964,A -85,B 0,C 180,E1 -13739.818,E2 -13739.818} C_VEL
LIN {X 0,Y 365.438,Z 281.05,A -85,B 0,C 180,E1 -13739.999,E2 -13739.999} C_VEL
LIN {X 0,Y 361.946,Z 404.552,A -85,B 0,C 180,E1 -13742.578,E2 -13742.578} C_VEL
LIN {X 0,Y 361.013,Z 419.931,A -85,B 0,C 180,E1 -13743.089,E2 -13743.089} C_VEL
LIN {X 0,Y 359.705,Z 434.93,A -85,B 0,C 180,E1 -13743.813,E2 -13743.813} C_VEL
LIN {X 0,Y 358.245,Z 449.247,A -85,B 0,C 180,E1 -13744.743,E2 -13744.743} C_VEL
LIN {X 0,Y 356.521,Z 462.79,A -85,B 0,C 180,E1 -13745.856,E2 -13745.856} C_VEL
LIN {X 0,Y 354.616,Z 476.546,A -85,B 0,C 180,E1 -13747.266,E2 -13747.266} C_VEL
LIN {X 0,Y 352.792,Z 488.988,A -85,B 0,C 180,E1 -13748.835,E2 -13748.835} C_VEL
LIN {X 0,Y 351.322,Z 499.452,A -85,B 0,C 180,E1 -13750.424,E2 -13750.424} C_VEL
LIN {X 0,Y 349.893,Z 509.104,A -85,B 0,C 180,E1 -13752.164,E2 -13752.164} C_VEL
LIN {X 0,Y 348.6,Z 518.581,A -85,B 0,C 180,E1 -13754.207,E2 -13754.207} C_VEL
LIN {X 0,Y 347.569,Z 526.335,A -85,B 0,C 180,E1 -13756.23,E2 -13756.23} C_VEL
LIN {X 0,Y 346.921,Z 532.9,A -85,B 0,C 180,E1 -13758.313,E2 -13758.313} C_VEL
LIN {X 0,Y 346.41,Z 538.811,A -85,B 0,C 180,E1 -13760.66,E2 -13760.66} C_VEL
LIN {X 0,Y 346.225,Z 543.292,A -85,B 0,C 180,E1 -13763.005,E2 -13763.005} C_VEL
LIN {X 0,Y 346.178,Z 546.438,A -85,B 0,C 180,E1 -13765.343,E2 -13765.343} C_VEL
LIN {X 0,Y 346.187,Z 548.313,A -85,B 0,C 180,E1 -13767.673,E2 -13767.673} C_VEL
LIN {X 0,Y 346.314,Z 548.951,A -85,B 0,C 180,E1 -13770,E2 -13770} C_VEL
LIN {X 0,Y 346.188,Z 548.304,A -85,B 0,C 180,E1 -13772.327,E2 -13772.327} C_VEL
LIN {X 0,Y 346.209,Z 546.421,A -85,B 0,C 180,E1 -13774.658,E2 -13774.658} C_VEL
LIN {X 0,Y 346.299,Z 543.273,A -85,B 0,C 180,E1 -13776.994,E2 -13776.994} C_VEL
LIN {X 0,Y 346.411,Z 538.785,A -85,B 0,C 180,E1 -13779.341,E2 -13779.341} C_VEL
LIN {X 0,Y 346.93,Z 532.859,A -85,B 0,C 180,E1 -13781.688,E2 -13781.688} C_VEL
LIN {X 0,Y 347.764,Z 525.238,A -85,B 0,C 180,E1 -13784.062,E2 -13784.062} C_VEL
LIN {X 0,Y 348.746,Z 517.247,A -85,B 0,C 180,E1 -13786.087,E2 -13786.087} C_VEL
LIN {X 0,Y 350.148,Z 507.507,A -85,B 0,C 180,E1 -13788.126,E2 -13788.126} C_VEL
LIN {X 0,Y 351.596,Z 497.538,A -85,B 0,C 180,E1 -13789.865,E2 -13789.865} C_VEL
LIN {X 0,Y 353.077,Z 486.742,A -85,B 0,C 180,E1 -13791.454,E2 -13791.454} C_VEL
LIN {X 0,Y 354.811,Z 475.129,A -85,B 0,C 180,E1 -13792.875,E2 -13792.875} C_VEL
LIN {X 0,Y 356.534,Z 462.612,A -85,B 0,C 180,E1 -13794.144,E2 -13794.144} C_VEL
LIN {X 0,Y 358.249,Z 449.017,A -85,B 0,C 180,E1 -13795.257,E2 -13795.257} C_VEL
LIN {X 0,Y 359.664,Z 435.173,A -85,B 0,C 180,E1 -13796.16,E2 -13796.16} C_VEL
LIN {X 0,Y 360.953,Z 420.437,A -85,B 0,C 180,E1 -13796.878,E2 -13796.878} C_VEL
LIN {X 0,Y 361.869,Z 405.336,A -85,B 0,C 180,E1 -13797.39,E2 -13797.39} C_VEL
LIN {X 0,Y 365.038,Z 294.53,A -85,B 0,C 180,E1 -13799.708,E2 -13799.708} C_VEL
LIN {X 0,Y 365.287,Z 280.122,A -85,B 0,C 180,E1 -13800.015,E2 -13800.015} C_VEL
LIN {X 0,Y 360.63,Z 251.266,A -85,B 0,C 180,E1 -13801.09,E2 -13801.09} C_VEL
LIN {X 0,Y 357.976,Z 244.905,A -85,B 0,C 180,E1 -13801.518,E2 -13801.518} C_VEL
LIN {X 0,Y 354.337,Z 230.764,A -85,B 0,C 180,E1 -13804.603,E2 -13804.603} C_VEL
LIN {X 0,Y 351.104,Z 219.475,A -85,B 0,C 180,E1 -13807.254,E2 -13807.254} C_VEL
LIN {X 0,Y 347.779,Z 208.881,A -85,B 0,C 180,E1 -13809.974,E2 -13809.974} C_VEL
LIN {X 0,Y 347.721,Z 208.792,A -85,B 0,C 180,E1 -13813.408,E2 -13813.408} C_VEL
LIN {X 0,Y 347.724,Z 208.792,A -85,B 0,C 180,E1 -13816.686,E2 -13816.686} C_VEL
LIN {X 0,Y 347.746,Z 208.797,A -85,B 0,C 180,E1 -13820.173,E2 -13820.173} C_VEL
LIN {X 0,Y 347.76,Z 208.776,A -85,B 0,C 180,E1 -13822.679,E2 -13822.679} C_VEL
LIN {X 0,Y 347.747,Z 208.785,A -85,B 0,C 180,E1 -13825.956,E2 -13825.956} C_VEL
LIN {X 0,Y 347.762,Z 208.789,A -85,B 0,C 180,E1 -13829.654,E2 -13829.654} C_VEL
LIN {X 0,Y 347.85,Z 208.753,A -85,B 0,C 180,E1 -13832.745,E2 -13832.745} C_VEL
LIN {X 0,Y 347.787,Z 208.787,A -85,B 0,C 180,E1 -13836.162,E2 -13836.162} C_VEL
LIN {X 0,Y 347.816,Z 208.784,A -85,B 0,C 180,E1 -13839.91,E2 -13839.91} C_VEL
LIN {X 0,Y 347.865,Z 208.772,A -85,B 0,C 180,E1 -13842.359,E2 -13842.359} C_VEL
LIN {X 0,Y 347.896,Z 208.767,A -85,B 0,C 180,E1 -13845.971,E2 -13845.971} C_VEL
LIN {X 0,Y 347.926,Z 208.766,A -85,B 0,C 180,E1 -13849.526,E2 -13849.526} C_VEL
LIN {X 0,Y 348.09,Z 208.749,A -85,B 0,C 180,E1 -13853.042,E2 -13853.042} C_VEL
LIN {X 0,Y 348.204,Z 208.732,A -85,B 0,C 180,E1 -13857.687,E2 -13857.687} C_VEL
LIN {X 0,Y 348.323,Z 208.719,A -85,B 0,C 180,E1 -13860,E2 -13860} C_VEL
LIN {X 0,Y 348.204,Z 208.73,A -85,B 0,C 180,E1 -13862.314,E2 -13862.314} C_VEL
LIN {X 0,Y 348.104,Z 208.743,A -85,B 0,C 180,E1 -13866.958,E2 -13866.958} C_VEL
LIN {X 0,Y 347.966,Z 208.765,A -85,B 0,C 180,E1 -13869.299,E2 -13869.299} C_VEL
LIN {X 0,Y 347.888,Z 208.769,A -85,B 0,C 180,E1 -13872.84,E2 -13872.84} C_VEL
LIN {X 0,Y 347.838,Z 208.773,A -85,B 0,C 180,E1 -13876.432,E2 -13876.432} C_VEL
LIN {X 0,Y 347.85,Z 208.779,A -85,B 0,C 180,E1 -13878.861,E2 -13878.861} C_VEL
LIN {X 0,Y 347.774,Z 208.79,A -85,B 0,C 180,E1 -13882.58,E2 -13882.58} C_VEL
LIN {X 0,Y 347.812,Z 208.786,A -85,B 0,C 180,E1 -13885.109,E2 -13885.109} C_VEL
LIN {X 0,Y 347.808,Z 208.765,A -85,B 0,C 180,E1 -13887.694,E2 -13887.694} C_VEL
LIN {X 0,Y 347.749,Z 208.781,A -85,B 0,C 180,E1 -13890.348,E2 -13890.348} C_VEL
LIN {X 0,Y 347.748,Z 208.774,A -85,B 0,C 180,E1 -13894.044,E2 -13894.044} C_VEL
LIN {X 0,Y 347.762,Z 208.792,A -85,B 0,C 180,E1 -13897.321,E2 -13897.321} C_VEL
LIN {X 0,Y 347.732,Z 208.777,A -85,B 0,C 180,E1 -13900.297,E2 -13900.297} C_VEL
LIN {X 0,Y 347.723,Z 208.786,A -85,B 0,C 180,E1 -13903.408,E2 -13903.408} C_VEL
LIN {X 0,Y 347.726,Z 208.792,A -85,B 0,C 180,E1 -13906.687,E2 -13906.687} C_VEL
LIN {X 0,Y 347.748,Z 208.787,A -85,B 0,C 180,E1 -13910.173,E2 -13910.173} C_VEL
LIN {X 0,Y 347.806,Z 208.978,A -85,B 0,C 180,E1 -13912.223,E2 -13912.223} C_VEL
LIN {X 0,Y 351.252,Z 220.898,A -85,B 0,C 180,E1 -13915.532,E2 -13915.532} C_VEL
LIN {X 0,Y 354.245,Z 232.69,A -85,B 0,C 180,E1 -13918.55,E2 -13918.55} C_VEL
LIN {X 0,Y 356.772,Z 243.839,A -85,B 0,C 180,E1 -13921.234,E2 -13921.234} C_VEL
LIN {X 0,Y 357.132,Z 245.212,A -85,B 0,C 180,E1 -13921.414,E2 -13921.414} C_VEL
LIN {X 0,Y 360.303,Z 258.77,A -85,B 0,C 180,E1 -13922.005,E2 -13922.005} C_VEL
LIN {X 0,Y 364.836,Z 282.292,A -85,B 0,C 180,E1 -13922.901,E2 -13922.901} C_VEL
LIN {X 0,Y 362.491,Z 388.305,A -85,B 0,C 180,E1 -13924.905,E2 -13924.905} C_VEL
LIN {X 0,Y 361.74,Z 402.763,A -85,B 0,C 180,E1 -13925.386,E2 -13925.386} C_VEL
LIN {X 0,Y 360.757,Z 416.545,A -85,B 0,C 180,E1 -13926.076,E2 -13926.076} C_VEL
LIN {X 0,Y 359.343,Z 429.991,A -85,B 0,C 180,E1 -13926.973,E2 -13926.973} C_VEL
LIN {X 0,Y 357.868,Z 442.843,A -85,B 0,C 180,E1 -13928.091,E2 -13928.091} C_VEL
LIN {X 0,Y 356.138,Z 454.525,A -85,B 0,C 180,E1 -13929.345,E2 -13929.345} C_VEL
LIN {X 0,Y 354.686,Z 464.255,A -85,B 0,C 180,E1 -13930.616,E2 -13930.616} C_VEL
LIN {X 0,Y 352.85,Z 475.007,A -85,B 0,C 180,E1 -13932.317,E2 -13932.317} C_VEL
LIN {X 0,Y 351.423,Z 483.93,A -85,B 0,C 180,E1 -13934.044,E2 -13934.044} C_VEL
LIN {X 0,Y 349.883,Z 492.439,A -85,B 0,C 180,E1 -13936.052,E2 -13936.052} C_VEL
LIN {X 0,Y 348.829,Z 498.492,A -85,B 0,C 180,E1 -13937.787,E2 -13937.787} C_VEL
LIN {X 0,Y 347.795,Z 504.931,A -85,B 0,C 180,E1 -13940.109,E2 -13940.109} C_VEL
LIN {X 0,Y 347.224,Z 508.75,A -85,B 0,C 180,E1 -13941.854,E2 -13941.854} C_VEL
LIN {X 0,Y 346.762,Z 512.561,A -85,B 0,C 180,E1 -13944.183,E2 -13944.183} C_VEL
LIN {X 0,Y 346.429,Z 515.049,A -85,B 0,C 180,E1 -13946.51,E2 -13946.51} C_VEL
LIN {X 0,Y 346.33,Z 516.287,A -85,B 0,C 180,E1 -13948.837,E2 -13948.837} C_VEL
LIN {X 0,Y 346.326,Z 516.313,A -85,B 0,C 180,E1 -13951.162,E2 -13951.162} C_VEL
LIN {X 0,Y 346.418,Z 515.133,A -85,B 0,C 180,E1 -13953.489,E2 -13953.489} C_VEL
LIN {X 0,Y 346.731,Z 512.706,A -85,B 0,C 180,E1 -13955.816,E2 -13955.816} C_VEL
LIN {X 0,Y 347.201,Z 508.958,A -85,B 0,C 180,E1 -13958.145,E2 -13958.145} C_VEL
LIN {X 0,Y 347.95,Z 503.759,A -85,B 0,C 180,E1 -13960.473,E2 -13960.473} C_VEL
LIN {X 0,Y 349.066,Z 496.934,A -85,B 0,C 180,E1 -13962.795,E2 -13962.795} C_VEL
LIN {X 0,Y 350.45,Z 489.422,A -85,B 0,C 180,E1 -13964.814,E2 -13964.814} C_VEL
LIN {X 0,Y 351.975,Z 480.183,A -85,B 0,C 180,E1 -13966.828,E2 -13966.828} C_VEL
LIN {X 0,Y 353.685,Z 470.513,A -85,B 0,C 180,E1 -13968.537,E2 -13968.537} C_VEL
LIN {X 0,Y 355.39,Z 459.805,A -85,B 0,C 180,E1 -13970.096,E2 -13970.096} C_VEL
LIN {X 0,Y 357.211,Z 447.958,A -85,B 0,C 180,E1 -13971.495,E2 -13971.495} C_VEL
LIN {X 0,Y 358.701,Z 436.358,A -85,B 0,C 180,E1 -13972.609,E2 -13972.609} C_VEL
LIN {X 0,Y 359.693,Z 427.53,A -85,B 0,C 180,E1 -13973.313,E2 -13973.313} C_VEL
LIN {X 0,Y 359.662,Z 422.203,A -85,B 0,C 180,E1 -13973.728,E2 -13973.728} C_VEL
LIN {X 0,Y 357.8,Z 413.556,A -85,B 0,C 180,E1 -13974.445,E2 -13974.445} C_VEL
LIN {X 0,Y 355.907,Z 404.711,A -85,B 0,C 180,E1 -13975.088,E2 -13975.088} C_VEL
LIN {X 0,Y 355.657,Z 399.082,A -85,B 0,C 180,E1 -13975.364,E2 -13975.364} C_VEL
LIN {X 0,Y 356.274,Z 384.501,A -85,B 0,C 180,E1 -13975.798,E2 -13975.798} C_VEL
LIN {X 0,Y 358.612,Z 282.631,A -85,B 0,C 180,E1 -13977.743,E2 -13977.743} C_VEL
LIN {X 0,Y 352.789,Z 253.593,A -85,B 0,C 180,E1 -13978.911,E2 -13978.911} C_VEL
LIN {X 0,Y 351.165,Z 247.724,A -85,B 0,C 180,E1 -13979.198,E2 -13979.198} C_VEL
LIN {X 0,Y 349.692,Z 244.238,A -85,B 0,C 180,E1 -13979.48,E2 -13979.48} C_VEL
LIN {X 0,Y 346.987,Z 232.225,A -85,B 0,C 180,E1 -13982.46,E2 -13982.46} C_VEL
LIN {X 0,Y 343.851,Z 220.215,A -85,B 0,C 180,E1 -13985.652,E2 -13985.652} C_VEL
LIN {X 0,Y 340.719,Z 209.758,A -85,B 0,C 180,E1 -13988.695,E2 -13988.695} C_VEL
LIN {X 0,Y 340.696,Z 209.66,A -85,B 0,C 180,E1 -13992.045,E2 -13992.045} C_VEL
LIN {X 0,Y 340.649,Z 209.664,A -85,B 0,C 180,E1 -13996.226,E2 -13996.226} C_VEL
LIN {X 0,Y 340.684,Z 209.656,A -85,B 0,C 180,E1 -13999.752,E2 -13999.752} C_VEL
LIN {X 0,Y 340.701,Z 209.67,A -85,B 0,C 180,E1 -14003.258,E2 -14003.258} C_VEL
LIN {X 0,Y 340.69,Z 209.654,A -85,B 0,C 180,E1 -14006.153,E2 -14006.153} C_VEL
LIN {X 0,Y 340.77,Z 209.639,A -85,B 0,C 180,E1 -14010.332,E2 -14010.332} C_VEL
LIN {X 0,Y 340.8,Z 209.645,A -85,B 0,C 180,E1 -14013.019,E2 -14013.019} C_VEL
LIN {X 0,Y 340.723,Z 209.662,A -85,B 0,C 180,E1 -14016.926,E2 -14016.926} C_VEL
LIN {X 0,Y 340.789,Z 209.653,A -85,B 0,C 180,E1 -14020.733,E2 -14020.733} C_VEL
LIN {X 0,Y 340.781,Z 209.654,A -85,B 0,C 180,E1 -14023.218,E2 -14023.218} C_VEL
LIN {X 0,Y 340.838,Z 209.651,A -85,B 0,C 180,E1 -14026.89,E2 -14026.89} C_VEL
LIN {X 0,Y 340.922,Z 209.646,A -85,B 0,C 180,E1 -14030.507,E2 -14030.507} C_VEL
LIN {X 0,Y 341.069,Z 209.618,A -85,B 0,C 180,E1 -14032.898,E2 -14032.898} C_VEL
LIN {X 0,Y 341.163,Z 209.606,A -85,B 0,C 180,E1 -14037.639,E2 -14037.639} C_VEL
LIN {X 0,Y 341.29,Z 209.595,A -85,B 0,C 180,E1 -14040,E2 -14040} C_VEL
LIN {X 0,Y 341.163,Z 209.608,A -85,B 0,C 180,E1 -14042.361,E2 -14042.361} C_VEL
LIN {X 0,Y 341.069,Z 209.624,A -85,B 0,C 180,E1 -14047.102,E2 -14047.102} C_VEL
LIN {X 0,Y 340.864,Z 209.647,A -85,B 0,C 180,E1 -14050.694,E2 -14050.694} C_VEL
LIN {X 0,Y 340.856,Z 209.644,A -85,B 0,C 180,E1 -14054.325,E2 -14054.325} C_VEL
LIN {X 0,Y 340.831,Z 209.65,A -85,B 0,C 180,E1 -14058.467,E2 -14058.467} C_VEL
LIN {X 0,Y 340.747,Z 209.659,A -85,B 0,C 180,E1 -14061.857,E2 -14061.857} C_VEL
LIN {X 0,Y 340.766,Z 209.637,A -85,B 0,C 180,E1 -14065.665,E2 -14065.665} C_VEL
LIN {X 0,Y 340.735,Z 209.655,A -85,B 0,C 180,E1 -14068.32,E2 -14068.32} C_VEL
LIN {X 0,Y 340.697,Z 209.66,A -85,B 0,C 180,E1 -14071.044,E2 -14071.044} C_VEL
LIN {X 0,Y 340.712,Z 209.672,A -85,B 0,C 180,E1 -14075.279,E2 -14075.279} C_VEL
LIN {X 0,Y 340.704,Z 209.656,A -85,B 0,C 180,E1 -14078.386,E2 -14078.386} C_VEL
LIN {X 0,Y 340.694,Z 209.656,A -85,B 0,C 180,E1 -14082.046,E2 -14082.046} C_VEL
LIN {X 0,Y 340.647,Z 209.668,A -85,B 0,C 180,E1 -14086.228,E2 -14086.228} C_VEL
LIN {X 0,Y 340.703,Z 209.847,A -85,B 0,C 180,E1 -14089.275,E2 -14089.275} C_VEL
LIN {X 0,Y 344.263,Z 221.035,A -85,B 0,C 180,E1 -14092.235,E2 -14092.235} C_VEL
LIN {X 0,Y 347.822,Z 233.442,A -85,B 0,C 180,E1 -14095.226,E2 -14095.226} C_VEL
LIN {X 0,Y 350.89,Z 245.151,A -85,B 0,C 180,E1 -14097.813,E2 -14097.813} C_VEL
LIN {X 0,Y 354.753,Z 254.083,A -85,B 0,C 180,E1 -14098.416,E2 -14098.416} C_VEL
LIN {X 0,Y 358.482,Z 277.143,A -85,B 0,C 180,E1 -14099.301,E2 -14099.301} C_VEL
LIN {X 0,Y 359.185,Z 283.676,A -85,B 0,C 180,E1 -14099.516,E2 -14099.516} C_VEL
LIN {X 0,Y 355.585,Z 404.892,A -85,B 0,C 180,E1 -14102.085,E2 -14102.085} C_VEL
LIN {X 0,Y 354.546,Z 420.901,A -85,B 0,C 180,E1 -14102.637,E2 -14102.637} C_VEL
LIN {X 0,Y 353.142,Z 436.03,A -85,B 0,C 180,E1 -14103.4,E2 -14103.4} C_VEL
LIN {X 0,Y 351.557,Z 450.712,A -85,B 0,C 180,E1 -14104.398,E2 -14104.398} C_VEL
LIN {X 0,Y 349.784,Z 463.844,A -85,B 0,C 180,E1 -14105.519,E2 -14105.519} C_VEL
LIN {X 0,Y 348.021,Z 476.13,A -85,B 0,C 180,E1 -14106.811,E2 -14106.811} C_VEL
LIN {X 0,Y 346.123,Z 488.599,A -85,B 0,C 180,E1 -14108.407,E2 -14108.407} C_VEL
LIN {X 0,Y 344.544,Z 499.069,A -85,B 0,C 180,E1 -14110.022,E2 -14110.022} C_VEL
LIN {X 0,Y 343.085,Z 508.737,A -85,B 0,C 180,E1 -14111.797,E2 -14111.797} C_VEL
LIN {X 0,Y 341.667,Z 518.221,A -85,B 0,C 180,E1 -14113.878,E2 -14113.878} C_VEL
LIN {X 0,Y 340.627,Z 525.719,A -85,B 0,C 180,E1 -14115.866,E2 -14115.866} C_VEL
LIN {X 0,Y 339.901,Z 532.555,A -85,B 0,C 180,E1 -14118.068,E2 -14118.068} C_VEL
LIN {X 0,Y 339.342,Z 538.471,A -85,B 0,C 180,E1 -14120.464,E2 -14120.464} C_VEL
LIN {X 0,Y 339.14,Z 542.956,A -85,B 0,C 180,E1 -14122.858,E2 -14122.858} C_VEL
LIN {X 0,Y 339.078,Z 546.103,A -85,B 0,C 180,E1 -14125.245,E2 -14125.245} C_VEL
LIN {X 0,Y 339.094,Z 547.979,A -85,B 0,C 180,E1 -14127.625,E2 -14127.625} C_VEL
LIN {X 0,Y 339.221,Z 548.618,A -85,B 0,C 180,E1 -14130,E2 -14130} C_VEL
LIN {X 0,Y 339.095,Z 547.971,A -85,B 0,C 180,E1 -14132.376,E2 -14132.376} C_VEL
LIN {X 0,Y 339.128,Z 546.086,A -85,B 0,C 180,E1 -14134.755,E2 -14134.755} C_VEL
LIN {X 0,Y 339.22,Z 542.935,A -85,B 0,C 180,E1 -14137.141,E2 -14137.141} C_VEL
LIN {X 0,Y 339.343,Z 538.442,A -85,B 0,C 180,E1 -14139.537,E2 -14139.537} C_VEL
LIN {X 0,Y 339.913,Z 532.511,A -85,B 0,C 180,E1 -14141.933,E2 -14141.933} C_VEL
LIN {X 0,Y 340.763,Z 524.978,A -85,B 0,C 180,E1 -14144.329,E2 -14144.329} C_VEL
LIN {X 0,Y 341.836,Z 516.885,A -85,B 0,C 180,E1 -14146.421,E2 -14146.421} C_VEL
LIN {X 0,Y 343.062,Z 508.654,A -85,B 0,C 180,E1 -14148.205,E2 -14148.205} C_VEL
LIN {X 0,Y 344.554,Z 498.968,A -85,B 0,C 180,E1 -14149.978,E2 -14149.978} C_VEL
LIN {X 0,Y 346.233,Z 487.421,A -85,B 0,C 180,E1 -14151.743,E2 -14151.743} C_VEL
LIN {X 0,Y 348.247,Z 474.698,A -85,B 0,C 180,E1 -14153.332,E2 -14153.332} C_VEL
LIN {X 0,Y 350.002,Z 462.14,A -85,B 0,C 180,E1 -14154.624,E2 -14154.624} C_VEL
LIN {X 0,Y 351.748,Z 448.901,A -85,B 0,C 180,E1 -14155.725,E2 -14155.725} C_VEL
LIN {X 0,Y 353.267,Z 434.557,A -85,B 0,C 180,E1 -14156.67,E2 -14156.67} C_VEL
LIN {X 0,Y 354.604,Z 419.659,A -85,B 0,C 180,E1 -14157.399,E2 -14157.399} C_VEL
LIN {X 0,Y 355.577,Z 404.201,A -85,B 0,C 180,E1 -14157.917,E2 -14157.917} C_VEL
LIN {X 0,Y 359.153,Z 282.799,A -85,B 0,C 180,E1 -14160.487,E2 -14160.487} C_VEL
LIN {X 0,Y 355.796,Z 260.42,A -85,B 0,C 180,E1 -14161.316,E2 -14161.316} C_VEL
LIN {X 0,Y 354.562,Z 253.666,A -85,B 0,C 180,E1 -14161.591,E2 -14161.591} C_VEL
LIN {X 0,Y 350.782,Z 244.896,A -85,B 0,C 180,E1 -14162.201,E2 -14162.201} C_VEL
LIN {X 0,Y 347.2,Z 231.201,A -85,B 0,C 180,E1 -14165.286,E2 -14165.286} C_VEL
LIN {X 0,Y 343.747,Z 219.301,A -85,B 0,C 180,E1 -14168.192,E2 -14168.192} C_VEL
LIN {X 0,Y 340.706,Z 209.774,A -85,B 0,C 180,E1 -14170.726,E2 -14170.726} C_VEL
LIN {X 0,Y 340.639,Z 209.667,A -85,B 0,C 180,E1 -14174.546,E2 -14174.546} C_VEL
LIN {X 0,Y 340.697,Z 209.656,A -85,B 0,C 180,E1 -14177.955,E2 -14177.955} C_VEL
LIN {X 0,Y 340.732,Z 209.652,A -85,B 0,C 180,E1 -14181.773,E2 -14181.773} C_VEL
LIN {X 0,Y 340.721,Z 209.667,A -85,B 0,C 180,E1 -14185.595,E2 -14185.595} C_VEL
LIN {X 0,Y 340.702,Z 209.659,A -85,B 0,C 180,E1 -14188.956,E2 -14188.956} C_VEL
LIN {X 0,Y 340.777,Z 209.637,A -85,B 0,C 180,E1 -14192.474,E2 -14192.474} C_VEL
LIN {X 0,Y 340.754,Z 209.658,A -85,B 0,C 180,E1 -14195.638,E2 -14195.638} C_VEL
LIN {X 0,Y 340.746,Z 209.661,A -85,B 0,C 180,E1 -14199.474,E2 -14199.474} C_VEL
LIN {X 0,Y 340.856,Z 209.645,A -85,B 0,C 180,E1 -14201.984,E2 -14201.984} C_VEL
LIN {X 0,Y 340.868,Z 209.643,A -85,B 0,C 180,E1 -14205.705,E2 -14205.705} C_VEL
LIN {X 0,Y 340.869,Z 209.647,A -85,B 0,C 180,E1 -14209.306,E2 -14209.306} C_VEL
LIN {X 0,Y 341.058,Z 209.625,A -85,B 0,C 180,E1 -14212.898,E2 -14212.898} C_VEL
LIN {X 0,Y 341.166,Z 209.609,A -85,B 0,C 180,E1 -14217.639,E2 -14217.639} C_VEL
LIN {X 0,Y 341.274,Z 209.596,A -85,B 0,C 180,E1 -14220,E2 -14220} C_VEL
LIN {X 0,Y 341.166,Z 209.606,A -85,B 0,C 180,E1 -14222.361,E2 -14222.361} C_VEL
LIN {X 0,Y 341.074,Z 209.617,A -85,B 0,C 180,E1 -14227.102,E2 -14227.102} C_VEL
LIN {X 0,Y 340.869,Z 209.649,A -85,B 0,C 180,E1 -14230.694,E2 -14230.694} C_VEL
LIN {X 0,Y 340.862,Z 209.649,A -85,B 0,C 180,E1 -14234.325,E2 -14234.325} C_VEL
LIN {X 0,Y 340.836,Z 209.653,A -85,B 0,C 180,E1 -14238.467,E2 -14238.467} C_VEL
LIN {X 0,Y 340.753,Z 209.664,A -85,B 0,C 180,E1 -14241.857,E2 -14241.857} C_VEL
LIN {X 0,Y 340.772,Z 209.661,A -85,B 0,C 180,E1 -14245.665,E2 -14245.665} C_VEL
LIN {X 0,Y 340.728,Z 209.64,A -85,B 0,C 180,E1 -14248.321,E2 -14248.321} C_VEL
LIN {X 0,Y 340.697,Z 209.667,A -85,B 0,C 180,E1 -14251.045,E2 -14251.045} C_VEL
LIN {X 0,Y 340.718,Z 209.647,A -85,B 0,C 180,E1 -14255.279,E2 -14255.279} C_VEL
LIN {X 0,Y 340.71,Z 209.663,A -85,B 0,C 180,E1 -14258.386,E2 -14258.386} C_VEL
LIN {X 0,Y 340.699,Z 209.672,A -85,B 0,C 180,E1 -14262.046,E2 -14262.046} C_VEL
LIN {X 0,Y 340.653,Z 209.679,A -85,B 0,C 180,E1 -14266.227,E2 -14266.227} C_VEL
LIN {X 0,Y 340.69,Z 209.671,A -85,B 0,C 180,E1 -14269.753,E2 -14269.753} C_VEL
LIN {X 0,Y 340.758,Z 209.871,A -85,B 0,C 180,E1 -14271.49,E2 -14271.49} C_VEL
LIN {X 0,Y 344.548,Z 222.76,A -85,B 0,C 180,E1 -14275.171,E2 -14275.171} C_VEL
LIN {X 0,Y 347.533,Z 234.649,A -85,B 0,C 180,E1 -14278.279,E2 -14278.279} C_VEL
LIN {X 0,Y 349.832,Z 244.608,A -85,B 0,C 180,E1 -14280.69,E2 -14280.69} C_VEL
LIN {X 0,Y 351.813,Z 249.547,A -85,B 0,C 180,E1 -14281.016,E2 -14281.016} C_VEL
LIN {X 0,Y 357.549,Z 277.031,A -85,B 0,C 180,E1 -14282.15,E2 -14282.15} C_VEL
LIN {X 0,Y 358.611,Z 283.204,A -85,B 0,C 180,E1 -14282.378,E2 -14282.378} C_VEL
LIN {X 0,Y 356.124,Z 389.33,A -85,B 0,C 180,E1 -14284.425,E2 -14284.425} C_VEL
LIN {X 0,Y 355.277,Z 404.232,A -85,B 0,C 180,E1 -14284.947,E2 -14284.947} C_VEL
LIN {X 0,Y 354.272,Z 417.518,A -85,B 0,C 180,E1 -14285.638,E2 -14285.638} C_VEL
LIN {X 0,Y 352.841,Z 430.484,A -85,B 0,C 180,E1 -14286.524,E2 -14286.524} C_VEL
LIN {X 0,Y 351.318,Z 443.286,A -85,B 0,C 180,E1 -14287.661,E2 -14287.661} C_VEL
LIN {X 0,Y 349.519,Z 454.936,A -85,B 0,C 180,E1 -14288.935,E2 -14288.935} C_VEL
LIN {X 0,Y 348.002,Z 464.643,A -85,B 0,C 180,E1 -14290.228,E2 -14290.228} C_VEL
LIN {X 0,Y 346.102,Z 475.378,A -85,B 0,C 180,E1 -14291.961,E2 -14291.961} C_VEL
LIN {X 0,Y 344.649,Z 483.838,A -85,B 0,C 180,E1 -14293.618,E2 -14293.618} C_VEL
LIN {X 0,Y 343.261,Z 491.703,A -85,B 0,C 180,E1 -14295.474,E2 -14295.474} C_VEL
LIN {X 0,Y 341.892,Z 498.836,A -85,B 0,C 180,E1 -14297.535,E2 -14297.535} C_VEL
LIN {X 0,Y 340.786,Z 505.273,A -85,B 0,C 180,E1 -14299.904,E2 -14299.904} C_VEL
LIN {X 0,Y 340.078,Z 510.143,A -85,B 0,C 180,E1 -14302.28,E2 -14302.28} C_VEL
LIN {X 0,Y 339.704,Z 512.897,A -85,B 0,C 180,E1 -14304.062,E2 -14304.062} C_VEL
LIN {X 0,Y 339.347,Z 515.383,A -85,B 0,C 180,E1 -14306.437,E2 -14306.437} C_VEL
LIN {X 0,Y 339.239,Z 516.62,A -85,B 0,C 180,E1 -14308.812,E2 -14308.812} C_VEL
LIN {X 0,Y 339.235,Z 516.646,A -85,B 0,C 180,E1 -14311.187,E2 -14311.187} C_VEL
LIN {X 0,Y 339.336,Z 515.466,A -85,B 0,C 180,E1 -14313.562,E2 -14313.562} C_VEL
LIN {X 0,Y 339.674,Z 513.04,A -85,B 0,C 180,E1 -14315.937,E2 -14315.937} C_VEL
LIN {X 0,Y 340.159,Z 509.295,A -85,B 0,C 180,E1 -14318.315,E2 -14318.315} C_VEL
LIN {X 0,Y 340.97,Z 504.1,A -85,B 0,C 180,E1 -14320.69,E2 -14320.69} C_VEL
LIN {X 0,Y 342.132,Z 497.28,A -85,B 0,C 180,E1 -14323.059,E2 -14323.059} C_VEL
LIN {X 0,Y 343.594,Z 489.774,A -85,B 0,C 180,E1 -14325.116,E2 -14325.116} C_VEL
LIN {X 0,Y 345.136,Z 480.831,A -85,B 0,C 180,E1 -14327.112,E2 -14327.112} C_VEL
LIN {X 0,Y 346.957,Z 470.887,A -85,B 0,C 180,E1 -14328.91,E2 -14328.91} C_VEL
LIN {X 0,Y 348.736,Z 460.197,A -85,B 0,C 180,E1 -14330.496,E2 -14330.496} C_VEL
LIN {X 0,Y 350.64,Z 448.375,A -85,B 0,C 180,E1 -14331.919,E2 -14331.919} C_VEL
LIN {X 0,Y 352.376,Z 435.575,A -85,B 0,C 180,E1 -14333.161,E2 -14333.161} C_VEL
LIN {X 0,Y 353.83,Z 422.152,A -85,B 0,C 180,E1 -14334.183,E2 -14334.183} C_VEL
LIN {X 0,Y 355.087,Z 407.906,A -85,B 0,C 180,E1 -14334.988,E2 -14334.988} C_VEL
LIN {X 0,Y 355.657,Z 399.082,A -85,B 0,C 180,E1 -14335.364,E2 -14335.364} C_VEL
LIN {X 0,Y 355.423,Z 393.374,A -85,B 0,C 180,E1 -14335.608,E2 -14335.608} C_VEL
LIN {X 0,Y 350.898,Z 374.806,A -85,B 0,C 180,E1 -14336.467,E2 -14336.467} C_VEL
LIN {X 0,Y 350.439,Z 369,A -85,B 0,C 180,E1 -14336.628,E2 -14336.628} C_VEL
LIN {X 0,Y 352.366,Z 283.707,A -85,B 0,C 180,E1 -14338.288,E2 -14338.288} C_VEL
LIN {X 0,Y 347.75,Z 260.278,A -85,B 0,C 180,E1 -14339.248,E2 -14339.248} C_VEL
LIN {X 0,Y 345.679,Z 251.313,A -85,B 0,C 180,E1 -14339.656,E2 -14339.656} C_VEL
LIN {X 0,Y 342.657,Z 244.587,A -85,B 0,C 180,E1 -14340.144,E2 -14340.144} C_VEL
LIN {X 0,Y 339.792,Z 232.37,A -85,B 0,C 180,E1 -14343.236,E2 -14343.236} C_VEL
LIN {X 0,Y 337.12,Z 222.172,A -85,B 0,C 180,E1 -14346.031,E2 -14346.031} C_VEL
LIN {X 0,Y 334.741,Z 214.243,A -85,B 0,C 180,E1 -14348.341,E2 -14348.341} C_VEL
LIN {X 0,Y 333.678,Z 210.628,A -85,B 0,C 180,E1 -14349.479,E2 -14349.479} C_VEL
LIN {X 0,Y 333.63,Z 210.54,A -85,B 0,C 180,E1 -14352.499,E2 -14352.499} C_VEL
LIN {X 0,Y 333.593,Z 210.542,A -85,B 0,C 180,E1 -14355.954,E2 -14355.954} C_VEL
LIN {X 0,Y 333.643,Z 210.537,A -85,B 0,C 180,E1 -14359.315,E2 -14359.315} C_VEL
LIN {X 0,Y 333.661,Z 210.548,A -85,B 0,C 180,E1 -14363.167,E2 -14363.167} C_VEL
LIN {X 0,Y 333.67,Z 210.524,A -85,B 0,C 180,E1 -14365.34,E2 -14365.34} C_VEL
LIN {X 0,Y 333.693,Z 210.532,A -85,B 0,C 180,E1 -14369.637,E2 -14369.637} C_VEL
LIN {X 0,Y 333.739,Z 210.515,A -85,B 0,C 180,E1 -14372.401,E2 -14372.401} C_VEL
LIN {X 0,Y 333.722,Z 210.539,A -85,B 0,C 180,E1 -14375.09,E2 -14375.09} C_VEL
LIN {X 0,Y 333.681,Z 210.542,A -85,B 0,C 180,E1 -14379.019,E2 -14379.019} C_VEL
LIN {X 0,Y 333.789,Z 210.531,A -85,B 0,C 180,E1 -14381.589,E2 -14381.589} C_VEL
LIN {X 0,Y 333.803,Z 210.529,A -85,B 0,C 180,E1 -14385.576,E2 -14385.576} C_VEL
LIN {X 0,Y 333.827,Z 210.522,A -85,B 0,C 180,E1 -14389.078,E2 -14389.078} C_VEL
LIN {X 0,Y 334.019,Z 210.495,A -85,B 0,C 180,E1 -14392.747,E2 -14392.747} C_VEL
LIN {X 0,Y 333.805,Z 210.528,A -85,B 0,C 180,E1 -14395.169,E2 -14395.169} C_VEL
LIN {X 0,Y 334.101,Z 210.486,A -85,B 0,C 180,E1 -14397.589,E2 -14397.589} C_VEL
LIN {X 0,Y 334.24,Z 210.473,A -85,B 0,C 180,E1 -14400,E2 -14400} C_VEL
LIN {X 0,Y 334.101,Z 210.489,A -85,B 0,C 180,E1 -14402.411,E2 -14402.411} C_VEL
LIN {X 0,Y 334.019,Z 210.502,A -85,B 0,C 180,E1 -14407.252,E2 -14407.252} C_VEL
LIN {X 0,Y 333.827,Z 210.525,A -85,B 0,C 180,E1 -14410.922,E2 -14410.922} C_VEL
LIN {X 0,Y 333.802,Z 210.525,A -85,B 0,C 180,E1 -14414.634,E2 -14414.634} C_VEL
LIN {X 0,Y 333.79,Z 210.528,A -85,B 0,C 180,E1 -14418.655,E2 -14418.655} C_VEL
LIN {X 0,Y 333.686,Z 210.541,A -85,B 0,C 180,E1 -14422.278,E2 -14422.278} C_VEL
LIN {X 0,Y 333.729,Z 210.508,A -85,B 0,C 180,E1 -14426.247,E2 -14426.247} C_VEL
LIN {X 0,Y 333.705,Z 210.54,A -85,B 0,C 180,E1 -14428.972,E2 -14428.972} C_VEL
LIN {X 0,Y 333.637,Z 210.525,A -85,B 0,C 180,E1 -14432.587,E2 -14432.587} C_VEL
LIN {X 0,Y 333.67,Z 210.541,A -85,B 0,C 180,E1 -14436.139,E2 -14436.139} C_VEL
LIN {X 0,Y 333.642,Z 210.546,A -85,B 0,C 180,E1 -14439.193,E2 -14439.193} C_VEL
LIN {X 0,Y 333.627,Z 210.538,A -85,B 0,C 180,E1 -14442.5,E2 -14442.5} C_VEL
LIN {X 0,Y 333.591,Z 210.545,A -85,B 0,C 180,E1 -14445.955,E2 -14445.955} C_VEL
LIN {X 0,Y 333.674,Z 210.761,A -85,B 0,C 180,E1 -14448.487,E2 -14448.487} C_VEL
LIN {X 0,Y 337.614,Z 223.128,A -85,B 0,C 180,E1 -14451.849,E2 -14451.849} C_VEL
LIN {X 0,Y 340.985,Z 234.819,A -85,B 0,C 180,E1 -14454.754,E2 -14454.754} C_VEL
LIN {X 0,Y 343.629,Z 245.07,A -85,B 0,C 180,E1 -14457.085,E2 -14457.085} C_VEL
LIN {X 0,Y 348.885,Z 256.808,A -85,B 0,C 180,E1 -14457.921,E2 -14457.921} C_VEL
LIN {X 0,Y 352.882,Z 282.317,A -85,B 0,C 180,E1 -14458.913,E2 -14458.913} C_VEL
LIN {X 0,Y 351.832,Z 321.453,A -85,B 0,C 180,E1 -14459.757,E2 -14459.757} C_VEL
LIN {X 0,Y 349.255,Z 405.211,A -85,B 0,C 180,E1 -14461.574,E2 -14461.574} C_VEL
LIN {X 0,Y 348.155,Z 420.988,A -85,B 0,C 180,E1 -14462.133,E2 -14462.133} C_VEL
LIN {X 0,Y 346.815,Z 435.119,A -85,B 0,C 180,E1 -14462.85,E2 -14462.85} C_VEL
LIN {X 0,Y 345.23,Z 449.335,A -85,B 0,C 180,E1 -14463.813,E2 -14463.813} C_VEL
LIN {X 0,Y 343.294,Z 463.405,A -85,B 0,C 180,E1 -14465.025,E2 -14465.025} C_VEL
LIN {X 0,Y 341.249,Z 476.919,A -85,B 0,C 180,E1 -14466.483,E2 -14466.483} C_VEL
LIN {X 0,Y 339.278,Z 489.204,A -85,B 0,C 180,E1 -14468.109,E2 -14468.109} C_VEL
LIN {X 0,Y 337.477,Z 500.667,A -85,B 0,C 180,E1 -14469.954,E2 -14469.954} C_VEL
LIN {X 0,Y 335.997,Z 509.866,A -85,B 0,C 180,E1 -14471.715,E2 -14471.715} C_VEL
LIN {X 0,Y 334.597,Z 519.107,A -85,B 0,C 180,E1 -14473.841,E2 -14473.841} C_VEL
LIN {X 0,Y 333.487,Z 526.719,A -85,B 0,C 180,E1 -14475.961,E2 -14475.961} C_VEL
LIN {X 0,Y 332.706,Z 533.873,A -85,B 0,C 180,E1 -14478.424,E2 -14478.424} C_VEL
LIN {X 0,Y 332.2,Z 539.42,A -85,B 0,C 180,E1 -14480.871,E2 -14480.871} C_VEL
LIN {X 0,Y 332.045,Z 542.618,A -85,B 0,C 180,E1 -14482.705,E2 -14482.705} C_VEL
LIN {X 0,Y 331.985,Z 545.769,A -85,B 0,C 180,E1 -14485.143,E2 -14485.143} C_VEL
LIN {X 0,Y 332.004,Z 547.647,A -85,B 0,C 180,E1 -14487.574,E2 -14487.574} C_VEL
LIN {X 0,Y 332.129,Z 548.285,A -85,B 0,C 180,E1 -14490,E2 -14490} C_VEL
LIN {X 0,Y 332.006,Z 547.638,A -85,B 0,C 180,E1 -14492.427,E2 -14492.427} C_VEL
LIN {X 0,Y 332.032,Z 545.751,A -85,B 0,C 180,E1 -14494.857,E2 -14494.857} C_VEL
LIN {X 0,Y 332.134,Z 542.596,A -85,B 0,C 180,E1 -14497.294,E2 -14497.294} C_VEL
LIN {X 0,Y 332.287,Z 538.1,A -85,B 0,C 180,E1 -14499.742,E2 -14499.742} C_VEL
LIN {X 0,Y 332.903,Z 532.165,A -85,B 0,C 180,E1 -14502.188,E2 -14502.188} C_VEL
LIN {X 0,Y 333.789,Z 524.624,A -85,B 0,C 180,E1 -14504.635,E2 -14504.635} C_VEL
LIN {X 0,Y 334.934,Z 516.523,A -85,B 0,C 180,E1 -14506.77,E2 -14506.77} C_VEL
LIN {X 0,Y 336.271,Z 508.284,A -85,B 0,C 180,E1 -14508.586,E2 -14508.586} C_VEL
LIN {X 0,Y 337.892,Z 498.087,A -85,B 0,C 180,E1 -14510.476,E2 -14510.476} C_VEL
LIN {X 0,Y 339.585,Z 487.017,A -85,B 0,C 180,E1 -14512.191,E2 -14512.191} C_VEL
LIN {X 0,Y 341.478,Z 475.572,A -85,B 0,C 180,E1 -14513.662,E2 -14513.662} C_VEL
LIN {X 0,Y 343.292,Z 463.227,A -85,B 0,C 180,E1 -14514.976,E2 -14514.976} C_VEL
LIN {X 0,Y 345.236,Z 449.165,A -85,B 0,C 180,E1 -14516.182,E2 -14516.182} C_VEL
LIN {X 0,Y 346.814,Z 434.828,A -85,B 0,C 180,E1 -14517.151,E2 -14517.151} C_VEL
LIN {X 0,Y 348.175,Z 420.624,A -85,B 0,C 180,E1 -14517.867,E2 -14517.867} C_VEL
LIN {X 0,Y 349.172,Z 405.813,A -85,B 0,C 180,E1 -14518.393,E2 -14518.393} C_VEL
LIN {X 0,Y 352.064,Z 312.619,A -85,B 0,C 180,E1 -14520.413,E2 -14520.413} C_VEL
LIN {X 0,Y 352.838,Z 282.056,A -85,B 0,C 180,E1 -14521.075,E2 -14521.075} C_VEL
LIN {X 0,Y 348.831,Z 256.692,A -85,B 0,C 180,E1 -14522.065,E2 -14522.065} C_VEL
LIN {X 0,Y 343.602,Z 244.933,A -85,B 0,C 180,E1 -14522.909,E2 -14522.909} C_VEL
LIN {X 0,Y 340.206,Z 231.876,A -85,B 0,C 180,E1 -14525.939,E2 -14525.939} C_VEL
LIN {X 0,Y 336.957,Z 220.804,A -85,B 0,C 180,E1 -14528.735,E2 -14528.735} C_VEL
LIN {X 0,Y 333.664,Z 210.645,A -85,B 0,C 180,E1 -14531.54,E2 -14531.54} C_VEL
LIN {X 0,Y 333.592,Z 210.555,A -85,B 0,C 180,E1 -14535.75,E2 -14535.75} C_VEL
LIN {X 0,Y 333.646,Z 210.545,A -85,B 0,C 180,E1 -14539.315,E2 -14539.315} C_VEL
LIN {X 0,Y 333.664,Z 210.534,A -85,B 0,C 180,E1 -14543.168,E2 -14543.168} C_VEL
LIN {X 0,Y 333.672,Z 210.547,A -85,B 0,C 180,E1 -14545.341,E2 -14545.341} C_VEL
LIN {X 0,Y 333.701,Z 210.541,A -85,B 0,C 180,E1 -14549.71,E2 -14549.71} C_VEL
LIN {X 0,Y 333.741,Z 210.513,A -85,B 0,C 180,E1 -14552.401,E2 -14552.401} C_VEL
LIN {X 0,Y 333.725,Z 210.525,A -85,B 0,C 180,E1 -14555.091,E2 -14555.091} C_VEL
LIN {X 0,Y 333.68,Z 210.54,A -85,B 0,C 180,E1 -14559.019,E2 -14559.019} C_VEL
LIN {X 0,Y 333.793,Z 210.526,A -85,B 0,C 180,E1 -14561.59,E2 -14561.59} C_VEL
LIN {X 0,Y 333.807,Z 210.523,A -85,B 0,C 180,E1 -14565.577,E2 -14565.577} C_VEL
LIN {X 0,Y 333.832,Z 210.525,A -85,B 0,C 180,E1 -14569.078,E2 -14569.078} C_VEL
LIN {X 0,Y 334.005,Z 210.504,A -85,B 0,C 180,E1 -14572.747,E2 -14572.747} C_VEL
LIN {X 0,Y 333.807,Z 210.521,A -85,B 0,C 180,E1 -14575.169,E2 -14575.169} C_VEL
LIN {X 0,Y 334.103,Z 210.489,A -85,B 0,C 180,E1 -14577.589,E2 -14577.589} C_VEL
LIN {X 0,Y 334.225,Z 210.474,A -85,B 0,C 180,E1 -14580,E2 -14580} C_VEL
LIN {X 0,Y 334.103,Z 210.486,A -85,B 0,C 180,E1 -14582.411,E2 -14582.411} C_VEL
LIN {X 0,Y 334.024,Z 210.494,A -85,B 0,C 180,E1 -14587.253,E2 -14587.253} C_VEL
LIN {X 0,Y 333.832,Z 210.523,A -85,B 0,C 180,E1 -14590.922,E2 -14590.922} C_VEL
LIN {X 0,Y 333.807,Z 210.529,A -85,B 0,C 180,E1 -14594.635,E2 -14594.635} C_VEL
LIN {X 0,Y 333.795,Z 210.531,A -85,B 0,C 180,E1 -14598.655,E2 -14598.655} C_VEL
LIN {X 0,Y 333.692,Z 210.543,A -85,B 0,C 180,E1 -14602.278,E2 -14602.278} C_VEL
LIN {X 0,Y 333.735,Z 210.538,A -85,B 0,C 180,E1 -14606.247,E2 -14606.247} C_VEL
LIN {X 0,Y 333.689,Z 210.515,A -85,B 0,C 180,E1 -14608.974,E2 -14608.974} C_VEL
LIN {X 0,Y 333.643,Z 210.548,A -85,B 0,C 180,E1 -14612.587,E2 -14612.587} C_VEL
LIN {X 0,Y 333.676,Z 210.534,A -85,B 0,C 180,E1 -14616.139,E2 -14616.139} C_VEL
LIN {X 0,Y 333.647,Z 210.532,A -85,B 0,C 180,E1 -14619.193,E2 -14619.193} C_VEL
LIN {X 0,Y 333.633,Z 210.551,A -85,B 0,C 180,E1 -14622.5,E2 -14622.5} C_VEL
LIN {X 0,Y 333.597,Z 210.557,A -85,B 0,C 180,E1 -14625.955,E2 -14625.955} C_VEL
LIN {X 0,Y 333.648,Z 210.552,A -85,B 0,C 180,E1 -14629.316,E2 -14629.316} C_VEL
LIN {X 0,Y 333.687,Z 210.771,A -85,B 0,C 180,E1 -14630.716,E2 -14630.716} C_VEL
LIN {X 0,Y 336.934,Z 221.655,A -85,B 0,C 180,E1 -14633.946,E2 -14633.946} C_VEL
LIN {X 0,Y 340.085,Z 233.358,A -85,B 0,C 180,E1 -14637.153,E2 -14637.153} C_VEL
LIN {X 0,Y 342.723,Z 244.629,A -85,B 0,C 180,E1 -14639.98,E2 -14639.98} C_VEL
LIN {X 0,Y 346.076,Z 252.543,A -85,B 0,C 180,E1 -14640.524,E2 -14640.524} C_VEL
LIN {X 0,Y 351.588,Z 279.656,A -85,B 0,C 180,E1 -14641.662,E2 -14641.662} C_VEL
LIN {X 0,Y 352.398,Z 284.309,A -85,B 0,C 180,E1 -14641.839,E2 -14641.839} C_VEL
LIN {X 0,Y 349.826,Z 389.105,A -85,B 0,C 180,E1 -14643.89,E2 -14643.89} C_VEL
LIN {X 0,Y 349.001,Z 403.386,A -85,B 0,C 180,E1 -14644.385,E2 -14644.385} C_VEL
LIN {X 0,Y 347.969,Z 416.841,A -85,B 0,C 180,E1 -14645.079,E2 -14645.079} C_VEL
LIN {X 0,Y 346.577,Z 429.223,A -85,B 0,C 180,E1 -14645.915,E2 -14645.915} C_VEL
LIN {X 0,Y 345.021,Z 442.343,A -85,B 0,C 180,E1 -14647.075,E2 -14647.075} C_VEL
LIN {X 0,Y 343.124,Z 454.188,A -85,B 0,C 180,E1 -14648.365,E2 -14648.365} C_VEL
LIN {X 0,Y 341.343,Z 465.03,A -85,B 0,C 180,E1 -14649.826,E2 -14649.826} C_VEL
LIN {X 0,Y 339.355,Z 475.75,A -85,B 0,C 180,E1 -14651.589,E2 -14651.589} C_VEL
LIN {X 0,Y 337.774,Z 484.504,A -85,B 0,C 180,E1 -14653.347,E2 -14653.347} C_VEL
LIN {X 0,Y 336.41,Z 492.052,A -85,B 0,C 180,E1 -14655.172,E2 -14655.172} C_VEL
LIN {X 0,Y 334.963,Z 499.18,A -85,B 0,C 180,E1 -14657.273,E2 -14657.273} C_VEL
LIN {X 0,Y 333.794,Z 505.613,A -85,B 0,C 180,E1 -14659.69,E2 -14659.69} C_VEL
LIN {X 0,Y 333.037,Z 510.48,A -85,B 0,C 180,E1 -14662.116,E2 -14662.116} C_VEL
LIN {X 0,Y 332.65,Z 513.233,A -85,B 0,C 180,E1 -14663.936,E2 -14663.936} C_VEL
LIN {X 0,Y 332.268,Z 515.717,A -85,B 0,C 180,E1 -14666.361,E2 -14666.361} C_VEL
LIN {X 0,Y 332.148,Z 516.953,A -85,B 0,C 180,E1 -14668.787,E2 -14668.787} C_VEL
LIN {X 0,Y 332.144,Z 516.979,A -85,B 0,C 180,E1 -14671.212,E2 -14671.212} C_VEL
LIN {X 0,Y 332.258,Z 515.799,A -85,B 0,C 180,E1 -14673.638,E2 -14673.638} C_VEL
LIN {X 0,Y 332.621,Z 513.373,A -85,B 0,C 180,E1 -14676.064,E2 -14676.064} C_VEL
LIN {X 0,Y 333.143,Z 509.631,A -85,B 0,C 180,E1 -14678.491,E2 -14678.491} C_VEL
LIN {X 0,Y 333.986,Z 504.44,A -85,B 0,C 180,E1 -14680.916,E2 -14680.916} C_VEL
LIN {X 0,Y 335.206,Z 497.624,A -85,B 0,C 180,E1 -14683.333,E2 -14683.333} C_VEL
LIN {X 0,Y 336.754,Z 490.124,A -85,B 0,C 180,E1 -14685.431,E2 -14685.431} C_VEL
LIN {X 0,Y 338.402,Z 480.901,A -85,B 0,C 180,E1 -14687.525,E2 -14687.525} C_VEL
LIN {X 0,Y 340.259,Z 471.259,A -85,B 0,C 180,E1 -14689.297,E2 -14689.297} C_VEL
LIN {X 0,Y 342.095,Z 460.588,A -85,B 0,C 180,E1 -14690.912,E2 -14690.912} C_VEL
LIN {X 0,Y 344.093,Z 448.79,A -85,B 0,C 180,E1 -14692.358,E2 -14692.358} C_VEL
LIN {X 0,Y 345.857,Z 436.29,A -85,B 0,C 180,E1 -14693.597,E2 -14693.597} C_VEL
LIN {X 0,Y 347.384,Z 422.683,A -85,B 0,C 180,E1 -14694.661,E2 -14694.661} C_VEL
LIN {X 0,Y 348.7,Z 408.578,A -85,B 0,C 180,E1 -14695.478,E2 -14695.478} C_VEL
LIN {X 0,Y 349.608,Z 394.694,A -85,B 0,C 180,E1 -14696.046,E2 -14696.046} C_VEL
LIN {X 0,Y 350.13,Z 380.706,A -85,B 0,C 180,E1 -14696.405,E2 -14696.405} C_VEL
LIN {X 0,Y 350.439,Z 369,A -85,B 0,C 180,E1 -14696.628,E2 -14696.628} C_VEL
LIN {X 0,Y 349.987,Z 363.192,A -85,B 0,C 180,E1 -14696.791,E2 -14696.791} C_VEL
LIN {X 0,Y 345.376,Z 344.536,A -85,B 0,C 180,E1 -14697.607,E2 -14697.607} C_VEL
LIN {X 0,Y 344.96,Z 338.728,A -85,B 0,C 180,E1 -14697.772,E2 -14697.772} C_VEL
LIN {X 0,Y 346.138,Z 284.408,A -85,B 0,C 180,E1 -14698.861,E2 -14698.861} C_VEL
LIN {X 0,Y 340.692,Z 256.833,A -85,B 0,C 180,E1 -14700.035,E2 -14700.035} C_VEL
LIN {X 0,Y 339.688,Z 253.702,A -85,B 0,C 180,E1 -14700.211,E2 -14700.211} C_VEL
LIN {X 0,Y 335.512,Z 244.52,A -85,B 0,C 180,E1 -14700.905,E2 -14700.905} C_VEL
LIN {X 0,Y 332.664,Z 232.442,A -85,B 0,C 180,E1 -14704.073,E2 -14704.073} C_VEL
LIN {X 0,Y 329.88,Z 222.313,A -85,B 0,C 180,E1 -14706.951,E2 -14706.951} C_VEL
LIN {X 0,Y 326.614,Z 211.485,A -85,B 0,C 180,E1 -14710.338,E2 -14710.338} C_VEL
LIN {X 0,Y 326.559,Z 211.429,A -85,B 0,C 180,E1 -14713.525,E2 -14713.525} C_VEL
LIN {X 0,Y 326.573,Z 211.424,A -85,B 0,C 180,E1 -14717.027,E2 -14717.027} C_VEL
LIN {X 0,Y 326.607,Z 211.409,A -85,B 0,C 180,E1 -14720.772,E2 -14720.772} C_VEL
LIN {X 0,Y 326.608,Z 211.407,A -85,B 0,C 180,E1 -14724.479,E2 -14724.479} C_VEL
LIN {X 0,Y 326.606,Z 211.423,A -85,B 0,C 180,E1 -14727.455,E2 -14727.455} C_VEL
LIN {X 0,Y 326.656,Z 211.395,A -85,B 0,C 180,E1 -14730.34,E2 -14730.34} C_VEL
LIN {X 0,Y 326.685,Z 211.416,A -85,B 0,C 180,E1 -14734.516,E2 -14734.516} C_VEL
LIN {X 0,Y 326.644,Z 211.423,A -85,B 0,C 180,E1 -14738.545,E2 -14738.545} C_VEL
LIN {X 0,Y 326.739,Z 211.407,A -85,B 0,C 180,E1 -14741.177,E2 -14741.177} C_VEL
LIN {X 0,Y 326.757,Z 211.408,A -85,B 0,C 180,E1 -14745.433,E2 -14745.433} C_VEL
LIN {X 0,Y 326.763,Z 211.4,A -85,B 0,C 180,E1 -14748.838,E2 -14748.838} C_VEL
LIN {X 0,Y 326.973,Z 211.372,A -85,B 0,C 180,E1 -14752.59,E2 -14752.59} C_VEL
LIN {X 0,Y 326.772,Z 211.404,A -85,B 0,C 180,E1 -14755.065,E2 -14755.065} C_VEL
LIN {X 0,Y 327.041,Z 211.365,A -85,B 0,C 180,E1 -14757.536,E2 -14757.536} C_VEL
LIN {X 0,Y 327.192,Z 211.35,A -85,B 0,C 180,E1 -14760,E2 -14760} C_VEL
LIN {X 0,Y 327.042,Z 211.368,A -85,B 0,C 180,E1 -14762.463,E2 -14762.463} C_VEL
LIN {X 0,Y 326.99,Z 211.37,A -85,B 0,C 180,E1 -14766.169,E2 -14766.169} C_VEL
LIN {X 0,Y 326.908,Z 211.384,A -85,B 0,C 180,E1 -14768.655,E2 -14768.655} C_VEL
LIN {X 0,Y 326.728,Z 211.409,A -85,B 0,C 180,E1 -14772.421,E2 -14772.421} C_VEL
LIN {X 0,Y 326.748,Z 211.406,A -85,B 0,C 180,E1 -14774.958,E2 -14774.958} C_VEL
LIN {X 0,Y 326.727,Z 211.409,A -85,B 0,C 180,E1 -14778.839,E2 -14778.839} C_VEL
LIN {X 0,Y 326.615,Z 211.425,A -85,B 0,C 180,E1 -14782.788,E2 -14782.788} C_VEL
LIN {X 0,Y 326.684,Z 211.391,A -85,B 0,C 180,E1 -14785.484,E2 -14785.484} C_VEL
LIN {X 0,Y 326.654,Z 211.423,A -85,B 0,C 180,E1 -14789.659,E2 -14789.659} C_VEL
LIN {X 0,Y 326.601,Z 211.414,A -85,B 0,C 180,E1 -14794.02,E2 -14794.02} C_VEL
LIN {X 0,Y 326.622,Z 211.406,A -85,B 0,C 180,E1 -14797.239,E2 -14797.239} C_VEL
LIN {X 0,Y 326.572,Z 211.419,A -85,B 0,C 180,E1 -14801.132,E2 -14801.132} C_VEL
LIN {X 0,Y 326.522,Z 211.428,A -85,B 0,C 180,E1 -14804.743,E2 -14804.743} C_VEL
LIN {X 0,Y 326.619,Z 211.628,A -85,B 0,C 180,E1 -14807.633,E2 -14807.633} C_VEL
LIN {X 0,Y 330.885,Z 224.68,A -85,B 0,C 180,E1 -14811.312,E2 -14811.312} C_VEL
LIN {X 0,Y 334.479,Z 237.425,A -85,B 0,C 180,E1 -14814.56,E2 -14814.56} C_VEL
LIN {X 0,Y 336.557,Z 245.271,A -85,B 0,C 180,E1 -14816.358,E2 -14816.358} C_VEL
LIN {X 0,Y 343.041,Z 259.578,A -85,B 0,C 180,E1 -14817.41,E2 -14817.41} C_VEL
LIN {X 0,Y 346.717,Z 283.421,A -85,B 0,C 180,E1 -14818.358,E2 -14818.358} C_VEL
LIN {X 0,Y 343.795,Z 381.362,A -85,B 0,C 180,E1 -14820.494,E2 -14820.494} C_VEL
LIN {X 0,Y 342.857,Z 406.59,A -85,B 0,C 180,E1 -14821.078,E2 -14821.078} C_VEL
LIN {X 0,Y 341.741,Z 421.832,A -85,B 0,C 180,E1 -14821.646,E2 -14821.646} C_VEL
LIN {X 0,Y 340.313,Z 436.046,A -85,B 0,C 180,E1 -14822.396,E2 -14822.396} C_VEL
LIN {X 0,Y 338.692,Z 449.841,A -85,B 0,C 180,E1 -14823.36,E2 -14823.36} C_VEL
LIN {X 0,Y 336.846,Z 462.967,A -85,B 0,C 180,E1 -14824.513,E2 -14824.513} C_VEL
LIN {X 0,Y 334.733,Z 476.513,A -85,B 0,C 180,E1 -14825.997,E2 -14825.997} C_VEL
LIN {X 0,Y 332.867,Z 487.821,A -85,B 0,C 180,E1 -14827.501,E2 -14827.501} C_VEL
LIN {X 0,Y 331.019,Z 498.675,A -85,B 0,C 180,E1 -14829.235,E2 -14829.235} C_VEL
LIN {X 0,Y 329.214,Z 509.506,A -85,B 0,C 180,E1 -14831.325,E2 -14831.325} C_VEL
LIN {X 0,Y 327.679,Z 518.753,A -85,B 0,C 180,E1 -14833.491,E2 -14833.491} C_VEL
LIN {X 0,Y 326.432,Z 526.915,A -85,B 0,C 180,E1 -14835.827,E2 -14835.827} C_VEL
LIN {X 0,Y 325.67,Z 533.529,A -85,B 0,C 180,E1 -14838.17,E2 -14838.17} C_VEL
LIN {X 0,Y 325.138,Z 539.08,A -85,B 0,C 180,E1 -14840.671,E2 -14840.671} C_VEL
LIN {X 0,Y 324.964,Z 542.281,A -85,B 0,C 180,E1 -14842.545,E2 -14842.545} C_VEL
LIN {X 0,Y 324.898,Z 545.435,A -85,B 0,C 180,E1 -14845.037,E2 -14845.037} C_VEL
LIN {X 0,Y 324.917,Z 547.314,A -85,B 0,C 180,E1 -14847.521,E2 -14847.521} C_VEL
LIN {X 0,Y 325.036,Z 547.953,A -85,B 0,C 180,E1 -14850,E2 -14850} C_VEL
LIN {X 0,Y 324.919,Z 547.305,A -85,B 0,C 180,E1 -14852.48,E2 -14852.48} C_VEL
LIN {X 0,Y 324.939,Z 545.416,A -85,B 0,C 180,E1 -14854.964,E2 -14854.964} C_VEL
LIN {X 0,Y 325.032,Z 542.257,A -85,B 0,C 180,E1 -14857.455,E2 -14857.455} C_VEL
LIN {X 0,Y 325.224,Z 537.758,A -85,B 0,C 180,E1 -14859.956,E2 -14859.956} C_VEL
LIN {X 0,Y 325.882,Z 531.818,A -85,B 0,C 180,E1 -14862.455,E2 -14862.455} C_VEL
LIN {X 0,Y 326.82,Z 524.271,A -85,B 0,C 180,E1 -14864.955,E2 -14864.955} C_VEL
LIN {X 0,Y 328.065,Z 516.163,A -85,B 0,C 180,E1 -14867.131,E2 -14867.131} C_VEL
LIN {X 0,Y 329.74,Z 506.393,A -85,B 0,C 180,E1 -14869.291,E2 -14869.291} C_VEL
LIN {X 0,Y 331.389,Z 496.379,A -85,B 0,C 180,E1 -14871.133,E2 -14871.133} C_VEL
LIN {X 0,Y 333.005,Z 486.616,A -85,B 0,C 180,E1 -14872.654,E2 -14872.654} C_VEL
LIN {X 0,Y 334.954,Z 475.145,A -85,B 0,C 180,E1 -14874.152,E2 -14874.152} C_VEL
LIN {X 0,Y 336.839,Z 462.777,A -85,B 0,C 180,E1 -14875.489,E2 -14875.489} C_VEL
LIN {X 0,Y 338.708,Z 449.618,A -85,B 0,C 180,E1 -14876.639,E2 -14876.639} C_VEL
LIN {X 0,Y 340.316,Z 435.762,A -85,B 0,C 180,E1 -14877.605,E2 -14877.605} C_VEL
LIN {X 0,Y 341.641,Z 422.206,A -85,B 0,C 180,E1 -14878.322,E2 -14878.322} C_VEL
LIN {X 0,Y 342.764,Z 407.121,A -85,B 0,C 180,E1 -14878.89,E2 -14878.89} C_VEL
LIN {X 0,Y 343.823,Z 378.759,A -85,B 0,C 180,E1 -14879.547,E2 -14879.547} C_VEL
LIN {X 0,Y 346.773,Z 284.172,A -85,B 0,C 180,E1 -14881.595,E2 -14881.595} C_VEL
LIN {X 0,Y 342.992,Z 259.338,A -85,B 0,C 180,E1 -14882.578,E2 -14882.578} C_VEL
LIN {X 0,Y 336.425,Z 244.893,A -85,B 0,C 180,E1 -14883.664,E2 -14883.664} C_VEL
LIN {X 0,Y 333.08,Z 232.292,A -85,B 0,C 180,E1 -14886.698,E2 -14886.698} C_VEL
LIN {X 0,Y 329.489,Z 220.368,A -85,B 0,C 180,E1 -14889.836,E2 -14889.836} C_VEL
LIN {X 0,Y 326.611,Z 211.539,A -85,B 0,C 180,E1 -14892.384,E2 -14892.384} C_VEL
LIN {X 0,Y 326.561,Z 211.431,A -85,B 0,C 180,E1 -14896.474,E2 -14896.474} C_VEL
LIN {X 0,Y 326.59,Z 211.431,A -85,B 0,C 180,E1 -14899.791,E2 -14899.791} C_VEL
LIN {X 0,Y 326.629,Z 211.408,A -85,B 0,C 180,E1 -14902.953,E2 -14902.953} C_VEL
LIN {X 0,Y 326.605,Z 211.416,A -85,B 0,C 180,E1 -14905.981,E2 -14905.981} C_VEL
LIN {X 0,Y 326.659,Z 211.423,A -85,B 0,C 180,E1 -14910.341,E2 -14910.341} C_VEL
LIN {X 0,Y 326.688,Z 211.391,A -85,B 0,C 180,E1 -14914.516,E2 -14914.516} C_VEL
LIN {X 0,Y 326.645,Z 211.414,A -85,B 0,C 180,E1 -14918.545,E2 -14918.545} C_VEL
LIN {X 0,Y 326.743,Z 211.407,A -85,B 0,C 180,E1 -14921.178,E2 -14921.178} C_VEL
LIN {X 0,Y 326.762,Z 211.402,A -85,B 0,C 180,E1 -14925.433,E2 -14925.433} C_VEL
LIN {X 0,Y 326.768,Z 211.404,A -85,B 0,C 180,E1 -14928.839,E2 -14928.839} C_VEL
LIN {X 0,Y 326.957,Z 211.382,A -85,B 0,C 180,E1 -14932.59,E2 -14932.59} C_VEL
LIN {X 0,Y 326.774,Z 211.396,A -85,B 0,C 180,E1 -14935.065,E2 -14935.065} C_VEL
LIN {X 0,Y 327.044,Z 211.369,A -85,B 0,C 180,E1 -14937.537,E2 -14937.537} C_VEL
LIN {X 0,Y 327.177,Z 211.351,A -85,B 0,C 180,E1 -14940,E2 -14940} C_VEL
LIN {X 0,Y 327.044,Z 211.365,A -85,B 0,C 180,E1 -14942.463,E2 -14942.463} C_VEL
LIN {X 0,Y 326.969,Z 211.373,A -85,B 0,C 180,E1 -14946.665,E2 -14946.665} C_VEL
LIN {X 0,Y 326.812,Z 211.401,A -85,B 0,C 180,E1 -14949.907,E2 -14949.907} C_VEL
LIN {X 0,Y 326.758,Z 211.409,A -85,B 0,C 180,E1 -14953.686,E2 -14953.686} C_VEL
LIN {X 0,Y 326.699,Z 211.416,A -85,B 0,C 180,E1 -14957.528,E2 -14957.528} C_VEL
LIN {X 0,Y 326.665,Z 211.41,A -85,B 0,C 180,E1 -14960.135,E2 -14960.135} C_VEL
LIN {X 0,Y 326.651,Z 211.414,A -85,B 0,C 180,E1 -14964.129,E2 -14964.129} C_VEL
LIN {X 0,Y 326.682,Z 211.405,A -85,B 0,C 180,E1 -14966.858,E2 -14966.858} C_VEL
LIN {X 0,Y 326.634,Z 211.413,A -85,B 0,C 180,E1 -14970.61,E2 -14970.61} C_VEL
LIN {X 0,Y 326.607,Z 211.406,A -85,B 0,C 180,E1 -14974.02,E2 -14974.02} C_VEL
LIN {X 0,Y 326.628,Z 211.426,A -85,B 0,C 180,E1 -14977.239,E2 -14977.239} C_VEL
LIN {X 0,Y 326.578,Z 211.419,A -85,B 0,C 180,E1 -14981.132,E2 -14981.132} C_VEL
LIN {X 0,Y 326.528,Z 211.423,A -85,B 0,C 180,E1 -14984.743,E2 -14984.743} C_VEL
LIN {X 0,Y 326.577,Z 211.418,A -85,B 0,C 180,E1 -14988.154,E2 -14988.154} C_VEL
LIN {X 0,Y 326.647,Z 211.577,A -85,B 0,C 180,E1 -14989.865,E2 -14989.865} C_VEL
LIN {X 0,Y 330.098,Z 223.108,A -85,B 0,C 180,E1 -14993.406,E2 -14993.406} C_VEL
LIN {X 0,Y 333.013,Z 233.906,A -85,B 0,C 180,E1 -14996.452,E2 -14996.452} C_VEL
LIN {X 0,Y 335.559,Z 244.64,A -85,B 0,C 180,E1 -14999.228,E2 -14999.228} C_VEL
LIN {X 0,Y 340.36,Z 255.509,A -85,B 0,C 180,E1 -15000.014,E2 -15000.014} C_VEL
LIN {X 0,Y 345.729,Z 282.381,A -85,B 0,C 180,E1 -15001.165,E2 -15001.165} C_VEL
LIN {X 0,Y 346.205,Z 285.653,A -85,B 0,C 180,E1 -15001.285,E2 -15001.285} C_VEL
LIN {X 0,Y 343.566,Z 388.831,A -85,B 0,C 180,E1 -15003.336,E2 -15003.336} C_VEL
LIN {X 0,Y 342.716,Z 403.308,A -85,B 0,C 180,E1 -15003.839,E2 -15003.839} C_VEL
LIN {X 0,Y 341.564,Z 417.406,A -85,B 0,C 180,E1 -15004.579,E2 -15004.579} C_VEL
LIN {X 0,Y 340.118,Z 429.883,A -85,B 0,C 180,E1 -15005.443,E2 -15005.443} C_VEL
LIN {X 0,Y 338.517,Z 442.843,A -85,B 0,C 180,E1 -15006.616,E2 -15006.616} C_VEL
LIN {X 0,Y 336.552,Z 454.597,A -85,B 0,C 180,E1 -15007.921,E2 -15007.921} C_VEL
LIN {X 0,Y 334.696,Z 465.416,A -85,B 0,C 180,E1 -15009.407,E2 -15009.407} C_VEL
LIN {X 0,Y 332.636,Z 476.12,A -85,B 0,C 180,E1 -15011.203,E2 -15011.203} C_VEL
LIN {X 0,Y 330.901,Z 485.291,A -85,B 0,C 180,E1 -15013.094,E2 -15013.094} C_VEL
LIN {X 0,Y 329.27,Z 493.49,A -85,B 0,C 180,E1 -15015.159,E2 -15015.159} C_VEL
LIN {X 0,Y 328.014,Z 499.526,A -85,B 0,C 180,E1 -15016.998,E2 -15016.998} C_VEL
LIN {X 0,Y 326.818,Z 505.952,A -85,B 0,C 180,E1 -15019.468,E2 -15019.468} C_VEL
LIN {X 0,Y 326.003,Z 510.817,A -85,B 0,C 180,E1 -15021.944,E2 -15021.944} C_VEL
LIN {X 0,Y 325.599,Z 513.568,A -85,B 0,C 180,E1 -15023.804,E2 -15023.804} C_VEL
LIN {X 0,Y 325.194,Z 516.051,A -85,B 0,C 180,E1 -15026.282,E2 -15026.282} C_VEL
LIN {X 0,Y 325.057,Z 517.286,A -85,B 0,C 180,E1 -15028.761,E2 -15028.761} C_VEL
LIN {X 0,Y 325.052,Z 517.311,A -85,B 0,C 180,E1 -15031.238,E2 -15031.238} C_VEL
LIN {X 0,Y 325.184,Z 516.131,A -85,B 0,C 180,E1 -15033.717,E2 -15033.717} C_VEL
LIN {X 0,Y 325.572,Z 513.706,A -85,B 0,C 180,E1 -15036.196,E2 -15036.196} C_VEL
LIN {X 0,Y 326.115,Z 509.967,A -85,B 0,C 180,E1 -15038.676,E2 -15038.676} C_VEL
LIN {X 0,Y 327.002,Z 504.78,A -85,B 0,C 180,E1 -15041.152,E2 -15041.152} C_VEL
LIN {X 0,Y 327.947,Z 499.838,A -85,B 0,C 180,E1 -15043.003,E2 -15043.003} C_VEL
LIN {X 0,Y 329.465,Z 492.786,A -85,B 0,C 180,E1 -15045.147,E2 -15045.147} C_VEL
LIN {X 0,Y 331.081,Z 484.127,A -85,B 0,C 180,E1 -15047.288,E2 -15047.288} C_VEL
LIN {X 0,Y 332.874,Z 475.079,A -85,B 0,C 180,E1 -15049.101,E2 -15049.101} C_VEL
LIN {X 0,Y 334.962,Z 464.132,A -85,B 0,C 180,E1 -15050.896,E2 -15050.896} C_VEL
LIN {X 0,Y 336.923,Z 453.032,A -85,B 0,C 180,E1 -15052.375,E2 -15052.375} C_VEL
LIN {X 0,Y 338.775,Z 441.281,A -85,B 0,C 180,E1 -15053.651,E2 -15053.651} C_VEL
LIN {X 0,Y 340.413,Z 428.456,A -85,B 0,C 180,E1 -15054.769,E2 -15054.769} C_VEL
LIN {X 0,Y 341.816,Z 415.185,A -85,B 0,C 180,E1 -15055.661,E2 -15055.661} C_VEL
LIN {X 0,Y 342.924,Z 401.279,A -85,B 0,C 180,E1 -15056.348,E2 -15056.348} C_VEL
LIN {X 0,Y 343.649,Z 386.858,A -85,B 0,C 180,E1 -15056.82,E2 -15056.82} C_VEL
LIN {X 0,Y 344.96,Z 338.728,A -85,B 0,C 180,E1 -15057.772,E2 -15057.772} C_VEL
LIN {X 0,Y 344.55,Z 332.921,A -85,B 0,C 180,E1 -15057.938,E2 -15057.938} C_VEL
LIN {X 0,Y 340.007,Z 314.28,A -85,B 0,C 180,E1 -15058.787,E2 -15058.787} C_VEL
LIN {X 0,Y 339.542,Z 308.476,A -85,B 0,C 180,E1 -15058.964,E2 -15058.964} C_VEL
LIN {X 0,Y 340.075,Z 285.915,A -85,B 0,C 180,E1 -15059.425,E2 -15059.425} C_VEL
LIN {X 0,Y 334.65,Z 258.199,A -85,B 0,C 180,E1 -15060.637,E2 -15060.637} C_VEL
LIN {X 0,Y 328.423,Z 244.668,A -85,B 0,C 180,E1 -15061.679,E2 -15061.679} C_VEL
LIN {X 0,Y 326.305,Z 235.682,A -85,B 0,C 180,E1 -15064.054,E2 -15064.054} C_VEL
LIN {X 0,Y 323.283,Z 224.57,A -85,B 0,C 180,E1 -15067.279,E2 -15067.279} C_VEL
LIN {X 0,Y 319.996,Z 213.935,A -85,B 0,C 180,E1 -15070.632,E2 -15070.632} C_VEL
LIN {X 0,Y 319.548,Z 212.358,A -85,B 0,C 180,E1 -15071.231,E2 -15071.231} C_VEL
LIN {X 0,Y 319.485,Z 212.306,A -85,B 0,C 180,E1 -15074.742,E2 -15074.742} C_VEL
LIN {X 0,Y 319.522,Z 212.31,A -85,B 0,C 180,E1 -15078.402,E2 -15078.402} C_VEL
LIN {X 0,Y 319.573,Z 212.305,A -85,B 0,C 180,E1 -15082.343,E2 -15082.343} C_VEL
LIN {X 0,Y 319.556,Z 212.281,A -85,B 0,C 180,E1 -15085.123,E2 -15085.123} C_VEL
LIN {X 0,Y 319.567,Z 212.297,A -85,B 0,C 180,E1 -15089.057,E2 -15089.057} C_VEL
LIN {X 0,Y 319.604,Z 212.275,A -85,B 0,C 180,E1 -15092.497,E2 -15092.497} C_VEL
LIN {X 0,Y 319.6,Z 212.296,A -85,B 0,C 180,E1 -15095.303,E2 -15095.303} C_VEL
LIN {X 0,Y 319.593,Z 212.299,A -85,B 0,C 180,E1 -15098.047,E2 -15098.047} C_VEL
LIN {X 0,Y 319.684,Z 212.283,A -85,B 0,C 180,E1 -15100.961,E2 -15100.961} C_VEL
LIN {X 0,Y 319.725,Z 212.282,A -85,B 0,C 180,E1 -15105.275,E2 -15105.275} C_VEL
LIN {X 0,Y 319.752,Z 212.279,A -85,B 0,C 180,E1 -15109.872,E2 -15109.872} C_VEL
LIN {X 0,Y 319.927,Z 212.249,A -85,B 0,C 180,E1 -15112.426,E2 -15112.426} C_VEL
LIN {X 0,Y 319.741,Z 212.281,A -85,B 0,C 180,E1 -15114.956,E2 -15114.956} C_VEL
LIN {X 0,Y 319.985,Z 212.243,A -85,B 0,C 180,E1 -15117.482,E2 -15117.482} C_VEL
LIN {X 0,Y 320.144,Z 212.228,A -85,B 0,C 180,E1 -15120,E2 -15120} C_VEL
LIN {X 0,Y 319.985,Z 212.248,A -85,B 0,C 180,E1 -15122.517,E2 -15122.517} C_VEL
LIN {X 0,Y 319.945,Z 212.248,A -85,B 0,C 180,E1 -15126.305,E2 -15126.305} C_VEL
LIN {X 0,Y 319.836,Z 212.264,A -85,B 0,C 180,E1 -15128.848,E2 -15128.848} C_VEL
LIN {X 0,Y 319.675,Z 212.286,A -85,B 0,C 180,E1 -15132.7,E2 -15132.7} C_VEL
LIN {X 0,Y 319.693,Z 212.285,A -85,B 0,C 180,E1 -15135.296,E2 -15135.296} C_VEL
LIN {X 0,Y 319.668,Z 212.289,A -85,B 0,C 180,E1 -15139.255,E2 -15139.255} C_VEL
LIN {X 0,Y 319.564,Z 212.304,A -85,B 0,C 180,E1 -15143.32,E2 -15143.32} C_VEL
LIN {X 0,Y 319.613,Z 212.266,A -85,B 0,C 180,E1 -15146.09,E2 -15146.09} C_VEL
LIN {X 0,Y 319.584,Z 212.299,A -85,B 0,C 180,E1 -15148.934,E2 -15148.934} C_VEL
LIN {X 0,Y 319.526,Z 212.284,A -85,B 0,C 180,E1 -15151.862,E2 -15151.862} C_VEL
LIN {X 0,Y 319.575,Z 212.302,A -85,B 0,C 180,E1 -15155.543,E2 -15155.543} C_VEL
LIN {X 0,Y 319.553,Z 212.307,A -85,B 0,C 180,E1 -15159.669,E2 -15159.669} C_VEL
LIN {X 0,Y 319.516,Z 212.307,A -85,B 0,C 180,E1 -15163.461,E2 -15163.461} C_VEL
LIN {X 0,Y 319.568,Z 212.521,A -85,B 0,C 180,E1 -15166.74,E2 -15166.74} C_VEL
LIN {X 0,Y 323.376,Z 224.042,A -85,B 0,C 180,E1 -15170.13,E2 -15170.13} C_VEL
LIN {X 0,Y 326.794,Z 235.625,A -85,B 0,C 180,E1 -15173.234,E2 -15173.234} C_VEL
LIN {X 0,Y 329.271,Z 244.92,A -85,B 0,C 180,E1 -15175.528,E2 -15175.528} C_VEL
LIN {X 0,Y 337.142,Z 261.921,A -85,B 0,C 180,E1 -15176.861,E2 -15176.861} C_VEL
LIN {X 0,Y 340.648,Z 284.97,A -85,B 0,C 180,E1 -15177.801,E2 -15177.801} C_VEL
LIN {X 0,Y 336.739,Z 404.483,A -85,B 0,C 180,E1 -15180.458,E2 -15180.458} C_VEL
LIN {X 0,Y 335.575,Z 420.416,A -85,B 0,C 180,E1 -15181.034,E2 -15181.034} C_VEL
LIN {X 0,Y 334.016,Z 435.497,A -85,B 0,C 180,E1 -15181.83,E2 -15181.83} C_VEL
LIN {X 0,Y 332.273,Z 449.726,A -85,B 0,C 180,E1 -15182.838,E2 -15182.838} C_VEL
LIN {X 0,Y 330.169,Z 463.97,A -85,B 0,C 180,E1 -15184.129,E2 -15184.129} C_VEL
LIN {X 0,Y 328.224,Z 476.108,A -85,B 0,C 180,E1 -15185.49,E2 -15185.49} C_VEL
LIN {X 0,Y 326.272,Z 487.431,A -85,B 0,C 180,E1 -15187.02,E2 -15187.02} C_VEL
LIN {X 0,Y 324.169,Z 499.09,A -85,B 0,C 180,E1 -15188.926,E2 -15188.926} C_VEL
LIN {X 0,Y 322.445,Z 509.145,A -85,B 0,C 180,E1 -15190.918,E2 -15190.918} C_VEL
LIN {X 0,Y 320.772,Z 518.398,A -85,B 0,C 180,E1 -15193.125,E2 -15193.125} C_VEL
LIN {X 0,Y 319.543,Z 526.24,A -85,B 0,C 180,E1 -15195.405,E2 -15195.405} C_VEL
LIN {X 0,Y 318.641,Z 533.185,A -85,B 0,C 180,E1 -15197.906,E2 -15197.906} C_VEL
LIN {X 0,Y 318.088,Z 538.741,A -85,B 0,C 180,E1 -15200.462,E2 -15200.462} C_VEL
LIN {X 0,Y 317.883,Z 541.944,A -85,B 0,C 180,E1 -15202.378,E2 -15202.378} C_VEL
LIN {X 0,Y 317.817,Z 545.101,A -85,B 0,C 180,E1 -15204.926,E2 -15204.926} C_VEL
LIN {X 0,Y 317.834,Z 546.981,A -85,B 0,C 180,E1 -15207.466,E2 -15207.466} C_VEL
LIN {X 0,Y 317.943,Z 547.62,A -85,B 0,C 180,E1 -15210,E2 -15210} C_VEL
LIN {X 0,Y 317.836,Z 546.972,A -85,B 0,C 180,E1 -15212.535,E2 -15212.535} C_VEL
LIN {X 0,Y 317.854,Z 545.081,A -85,B 0,C 180,E1 -15215.074,E2 -15215.074} C_VEL
LIN {X 0,Y 317.953,Z 541.919,A -85,B 0,C 180,E1 -15217.622,E2 -15217.622} C_VEL
LIN {X 0,Y 318.152,Z 537.415,A -85,B 0,C 180,E1 -15220.179,E2 -15220.179} C_VEL
LIN {X 0,Y 318.858,Z 531.47,A -85,B 0,C 180,E1 -15222.734,E2 -15222.734} C_VEL
LIN {X 0,Y 319.897,Z 523.919,A -85,B 0,C 180,E1 -15225.286,E2 -15225.286} C_VEL
LIN {X 0,Y 321.203,Z 515.803,A -85,B 0,C 180,E1 -15227.509,E2 -15227.509} C_VEL
LIN {X 0,Y 322.936,Z 506.021,A -85,B 0,C 180,E1 -15229.714,E2 -15229.714} C_VEL
LIN {X 0,Y 324.685,Z 495.995,A -85,B 0,C 180,E1 -15231.591,E2 -15231.591} C_VEL
LIN {X 0,Y 326.418,Z 486.215,A -85,B 0,C 180,E1 -15233.137,E2 -15233.137} C_VEL
LIN {X 0,Y 328.442,Z 474.717,A -85,B 0,C 180,E1 -15234.662,E2 -15234.662} C_VEL
LIN {X 0,Y 330.407,Z 462.323,A -85,B 0,C 180,E1 -15236.022,E2 -15236.022} C_VEL
LIN {X 0,Y 332.351,Z 448.759,A -85,B 0,C 180,E1 -15237.223,E2 -15237.223} C_VEL
LIN {X 0,Y 334.147,Z 433.998,A -85,B 0,C 180,E1 -15238.245,E2 -15238.245} C_VEL
LIN {X 0,Y 335.621,Z 419.131,A -85,B 0,C 180,E1 -15239.006,E2 -15239.006} C_VEL
LIN {X 0,Y 336.719,Z 403.689,A -85,B 0,C 180,E1 -15239.545,E2 -15239.545} C_VEL
LIN {X 0,Y 340.626,Z 285.14,A -85,B 0,C 180,E1 -15242.173,E2 -15242.173} C_VEL
LIN {X 0,Y 337.132,Z 262,A -85,B 0,C 180,E1 -15243.113,E2 -15243.113} C_VEL
LIN {X 0,Y 329.273,Z 244.973,A -85,B 0,C 180,E1 -15244.438,E2 -15244.438} C_VEL
LIN {X 0,Y 325.991,Z 232.718,A -85,B 0,C 180,E1 -15247.492,E2 -15247.492} C_VEL
LIN {X 0,Y 322.786,Z 222.207,A -85,B 0,C 180,E1 -15250.355,E2 -15250.355} C_VEL
LIN {X 0,Y 319.535,Z 212.433,A -85,B 0,C 180,E1 -15253.277,E2 -15253.277} C_VEL
LIN {X 0,Y 319.553,Z 212.295,A -85,B 0,C 180,E1 -15257.017,E2 -15257.017} C_VEL
LIN {X 0,Y 319.546,Z 212.308,A -85,B 0,C 180,E1 -15260.371,E2 -15260.371} C_VEL
LIN {X 0,Y 319.579,Z 212.304,A -85,B 0,C 180,E1 -15264.457,E2 -15264.457} C_VEL
LIN {X 0,Y 319.53,Z 212.284,A -85,B 0,C 180,E1 -15268.138,E2 -15268.138} C_VEL
LIN {X 0,Y 319.615,Z 212.284,A -85,B 0,C 180,E1 -15271.589,E2 -15271.589} C_VEL
LIN {X 0,Y 319.603,Z 212.286,A -85,B 0,C 180,E1 -15275.304,E2 -15275.304} C_VEL
LIN {X 0,Y 319.596,Z 212.294,A -85,B 0,C 180,E1 -15278.048,E2 -15278.048} C_VEL
LIN {X 0,Y 319.688,Z 212.286,A -85,B 0,C 180,E1 -15280.962,E2 -15280.962} C_VEL
LIN {X 0,Y 319.729,Z 212.279,A -85,B 0,C 180,E1 -15285.276,E2 -15285.276} C_VEL
LIN {X 0,Y 319.751,Z 212.272,A -85,B 0,C 180,E1 -15289.873,E2 -15289.873} C_VEL
LIN {X 0,Y 319.911,Z 212.26,A -85,B 0,C 180,E1 -15292.426,E2 -15292.426} C_VEL
LIN {X 0,Y 319.744,Z 212.271,A -85,B 0,C 180,E1 -15294.956,E2 -15294.956} C_VEL
LIN {X 0,Y 319.988,Z 212.248,A -85,B 0,C 180,E1 -15297.483,E2 -15297.483} C_VEL
LIN {X 0,Y 320.129,Z 212.229,A -85,B 0,C 180,E1 -15300,E2 -15300} C_VEL
LIN {X 0,Y 319.988,Z 212.244,A -85,B 0,C 180,E1 -15302.518,E2 -15302.518} C_VEL
LIN {X 0,Y 319.93,Z 212.251,A -85,B 0,C 180,E1 -15306.656,E2 -15306.656} C_VEL
LIN {X 0,Y 319.757,Z 212.279,A -85,B 0,C 180,E1 -15310.127,E2 -15310.127} C_VEL
LIN {X 0,Y 319.73,Z 212.282,A -85,B 0,C 180,E1 -15314.724,E2 -15314.724} C_VEL
LIN {X 0,Y 319.688,Z 212.283,A -85,B 0,C 180,E1 -15319.038,E2 -15319.038} C_VEL
LIN {X 0,Y 319.57,Z 212.296,A -85,B 0,C 180,E1 -15323.32,E2 -15323.32} C_VEL
LIN {X 0,Y 319.634,Z 212.294,A -85,B 0,C 180,E1 -15326.088,E2 -15326.088} C_VEL
LIN {X 0,Y 319.579,Z 212.271,A -85,B 0,C 180,E1 -15328.935,E2 -15328.935} C_VEL
LIN {X 0,Y 319.53,Z 212.308,A -85,B 0,C 180,E1 -15331.862,E2 -15331.862} C_VEL
LIN {X 0,Y 319.58,Z 212.28,A -85,B 0,C 180,E1 -15335.543,E2 -15335.543} C_VEL
LIN {X 0,Y 319.573,Z 212.301,A -85,B 0,C 180,E1 -15338.008,E2 -15338.008} C_VEL
LIN {X 0,Y 319.526,Z 212.306,A -85,B 0,C 180,E1 -15341.597,E2 -15341.597} C_VEL
LIN {X 0,Y 319.489,Z 212.304,A -85,B 0,C 180,E1 -15345.257,E2 -15345.257} C_VEL
LIN {X 0,Y 319.531,Z 212.315,A -85,B 0,C 180,E1 -15348.712,E2 -15348.712} C_VEL
LIN {X 0,Y 319.579,Z 212.543,A -85,B 0,C 180,E1 -15349.025,E2 -15349.025} C_VEL
LIN {X 0,Y 322.482,Z 221.96,A -85,B 0,C 180,E1 -15352.047,E2 -15352.047} C_VEL
LIN {X 0,Y 325.782,Z 233.707,A -85,B 0,C 180,E1 -15355.512,E2 -15355.512} C_VEL
LIN {X 0,Y 328.177,Z 243.741,A -85,B 0,C 180,E1 -15358.251,E2 -15358.251} C_VEL
LIN {X 0,Y 328.641,Z 245.272,A -85,B 0,C 180,E1 -15358.495,E2 -15358.495} C_VEL
LIN {X 0,Y 334.555,Z 257.964,A -85,B 0,C 180,E1 -15359.462,E2 -15359.462} C_VEL
LIN {X 0,Y 339.91,Z 285.393,A -85,B 0,C 180,E1 -15360.66,E2 -15360.66} C_VEL
LIN {X 0,Y 339.392,Z 312.346,A -85,B 0,C 180,E1 -15361.221,E2 -15361.221} C_VEL
LIN {X 0,Y 337.28,Z 389.854,A -85,B 0,C 180,E1 -15362.799,E2 -15362.799} C_VEL
LIN {X 0,Y 336.331,Z 404.77,A -85,B 0,C 180,E1 -15363.345,E2 -15363.345} C_VEL
LIN {X 0,Y 335.198,Z 417.967,A -85,B 0,C 180,E1 -15364.061,E2 -15364.061} C_VEL
LIN {X 0,Y 333.731,Z 430.211,A -85,B 0,C 180,E1 -15364.926,E2 -15364.926} C_VEL
LIN {X 0,Y 332.038,Z 443.32,A -85,B 0,C 180,E1 -15366.136,E2 -15366.136} C_VEL
LIN {X 0,Y 330.009,Z 455.004,A -85,B 0,C 180,E1 -15367.459,E2 -15367.459} C_VEL
LIN {X 0,Y 328.044,Z 465.803,A -85,B 0,C 180,E1 -15368.97,E2 -15368.97} C_VEL
LIN {X 0,Y 325.939,Z 476.489,A -85,B 0,C 180,E1 -15370.802,E2 -15370.802} C_VEL
LIN {X 0,Y 324.043,Z 485.953,A -85,B 0,C 180,E1 -15372.8,E2 -15372.8} C_VEL
LIN {X 0,Y 322.42,Z 493.839,A -85,B 0,C 180,E1 -15374.836,E2 -15374.836} C_VEL
LIN {X 0,Y 321.083,Z 499.87,A -85,B 0,C 180,E1 -15376.713,E2 -15376.713} C_VEL
LIN {X 0,Y 319.821,Z 506.293,A -85,B 0,C 180,E1 -15379.234,E2 -15379.234} C_VEL
LIN {X 0,Y 318.974,Z 511.154,A -85,B 0,C 180,E1 -15381.766,E2 -15381.766} C_VEL
LIN {X 0,Y 318.551,Z 513.903,A -85,B 0,C 180,E1 -15383.666,E2 -15383.666} C_VEL
LIN {X 0,Y 318.124,Z 516.384,A -85,B 0,C 180,E1 -15386.199,E2 -15386.199} C_VEL
LIN {X 0,Y 317.967,Z 517.619,A -85,B 0,C 180,E1 -15388.733,E2 -15388.733} C_VEL
LIN {X 0,Y 317.961,Z 517.644,A -85,B 0,C 180,E1 -15391.266,E2 -15391.266} C_VEL
LIN {X 0,Y 318.113,Z 516.464,A -85,B 0,C 180,E1 -15393.8,E2 -15393.8} C_VEL
LIN {X 0,Y 318.526,Z 514.039,A -85,B 0,C 180,E1 -15396.333,E2 -15396.333} C_VEL
LIN {X 0,Y 319.108,Z 510.301,A -85,B 0,C 180,E1 -15398.868,E2 -15398.868} C_VEL
LIN {X 0,Y 320.037,Z 505.119,A -85,B 0,C 180,E1 -15401.398,E2 -15401.398} C_VEL
LIN {X 0,Y 321.382,Z 498.313,A -85,B 0,C 180,E1 -15403.918,E2 -15403.918} C_VEL
LIN {X 0,Y 323.102,Z 490.823,A -85,B 0,C 180,E1 -15406.1,E2 -15406.1} C_VEL
LIN {X 0,Y 324.601,Z 483.07,A -85,B 0,C 180,E1 -15407.97,E2 -15407.97} C_VEL
LIN {X 0,Y 326.55,Z 473.752,A -85,B 0,C 180,E1 -15409.813,E2 -15409.813} C_VEL
LIN {X 0,Y 328.529,Z 463.471,A -85,B 0,C 180,E1 -15411.489,E2 -15411.489} C_VEL
LIN {X 0,Y 330.591,Z 452.171,A -85,B 0,C 180,E1 -15412.993,E2 -15412.993} C_VEL
LIN {X 0,Y 332.482,Z 440.501,A -85,B 0,C 180,E1 -15414.257,E2 -15414.257} C_VEL
LIN {X 0,Y 334.123,Z 427.773,A -85,B 0,C 180,E1 -15415.367,E2 -15415.367} C_VEL
LIN {X 0,Y 335.579,Z 414.475,A -85,B 0,C 180,E1 -15416.257,E2 -15416.257} C_VEL
LIN {X 0,Y 336.742,Z 400.182,A -85,B 0,C 180,E1 -15416.954,E2 -15416.954} C_VEL
LIN {X 0,Y 337.435,Z 386.455,A -85,B 0,C 180,E1 -15417.397,E2 -15417.397} C_VEL
LIN {X 0,Y 339.542,Z 308.476,A -85,B 0,C 180,E1 -15418.964,E2 -15418.964} C_VEL
LIN {X 0,Y 339.087,Z 302.659,A -85,B 0,C 180,E1 -15419.142,E2 -15419.142} C_VEL
LIN {X 0,Y 336.691,Z 293.391,A -85,B 0,C 180,E1 -15419.596,E2 -15419.596} C_VEL
LIN {X 0,Y 334.3,Z 286.082,A -85,B 0,C 180,E1 -15420.014,E2 -15420.014} C_VEL
LIN {X 0,Y 332.453,Z 278.562,A -85,B 0,C 180,E1 -15420.386,E2 -15420.386} C_VEL
LIN {X 0,Y 328.747,Z 260.563,A -85,B 0,C 180,E1 -15421.226,E2 -15421.226} C_VEL
LIN {X 0,Y 321.267,Z 244.561,A -85,B 0,C 180,E1 -15422.525,E2 -15422.525} C_VEL
LIN {X 0,Y 318.403,Z 232.906,A -85,B 0,C 180,E1 -15425.79,E2 -15425.79} C_VEL
LIN {X 0,Y 315.586,Z 223.174,A -85,B 0,C 180,E1 -15428.79,E2 -15428.79} C_VEL
LIN {X 0,Y 312.498,Z 213.323,A -85,B 0,C 180,E1 -15432.084,E2 -15432.084} C_VEL
LIN {X 0,Y 312.455,Z 213.174,A -85,B 0,C 180,E1 -15436.034,E2 -15436.034} C_VEL
LIN {X 0,Y 312.5,Z 213.164,A -85,B 0,C 180,E1 -15439.874,E2 -15439.874} C_VEL
LIN {X 0,Y 312.533,Z 213.183,A -85,B 0,C 180,E1 -15442.616,E2 -15442.616} C_VEL
LIN {X 0,Y 312.515,Z 213.162,A -85,B 0,C 180,E1 -15446.31,E2 -15446.31} C_VEL
LIN {X 0,Y 312.541,Z 213.152,A -85,B 0,C 180,E1 -15450.349,E2 -15450.349} C_VEL
LIN {X 0,Y 312.598,Z 213.17,A -85,B 0,C 180,E1 -15454.064,E2 -15454.064} C_VEL
LIN {X 0,Y 312.582,Z 213.172,A -85,B 0,C 180,E1 -15457.528,E2 -15457.528} C_VEL
LIN {X 0,Y 312.633,Z 213.167,A -85,B 0,C 180,E1 -15461.656,E2 -15461.656} C_VEL
LIN {X 0,Y 312.688,Z 213.16,A -85,B 0,C 180,E1 -15465.686,E2 -15465.686} C_VEL
LIN {X 0,Y 312.696,Z 213.158,A -85,B 0,C 180,E1 -15469.641,E2 -15469.641} C_VEL
LIN {X 0,Y 312.866,Z 213.128,A -85,B 0,C 180,E1 -15472.254,E2 -15472.254} C_VEL
LIN {X 0,Y 312.712,Z 213.157,A -85,B 0,C 180,E1 -15474.842,E2 -15474.842} C_VEL
LIN {X 0,Y 312.984,Z 213.125,A -85,B 0,C 180,E1 -15478.713,E2 -15478.713} C_VEL
LIN {X 0,Y 312.984,Z 213.111,A -85,B 0,C 180,E1 -15481.286,E2 -15481.286} C_VEL
LIN {X 0,Y 312.712,Z 213.146,A -85,B 0,C 180,E1 -15485.157,E2 -15485.157} C_VEL
LIN {X 0,Y 312.865,Z 213.139,A -85,B 0,C 180,E1 -15487.746,E2 -15487.746} C_VEL
LIN {X 0,Y 312.663,Z 213.163,A -85,B 0,C 180,E1 -15491.671,E2 -15491.671} C_VEL
LIN {X 0,Y 312.694,Z 213.156,A -85,B 0,C 180,E1 -15494.888,E2 -15494.888} C_VEL
LIN {X 0,Y 312.624,Z 213.166,A -85,B 0,C 180,E1 -15499.237,E2 -15499.237} C_VEL
LIN {X 0,Y 312.54,Z 213.178,A -85,B 0,C 180,E1 -15502.789,E2 -15502.789} C_VEL
LIN {X 0,Y 312.591,Z 213.141,A -85,B 0,C 180,E1 -15505.934,E2 -15505.934} C_VEL
LIN {X 0,Y 312.539,Z 213.181,A -85,B 0,C 180,E1 -15509.65,E2 -15509.65} C_VEL
LIN {X 0,Y 312.514,Z 213.162,A -85,B 0,C 180,E1 -15513.689,E2 -15513.689} C_VEL
LIN {X 0,Y 312.515,Z 213.161,A -85,B 0,C 180,E1 -15517.386,E2 -15517.386} C_VEL
LIN {X 0,Y 312.485,Z 213.178,A -85,B 0,C 180,E1 -15520.71,E2 -15520.71} C_VEL
LIN {X 0,Y 312.446,Z 213.188,A -85,B 0,C 180,E1 -15524.21,E2 -15524.21} C_VEL
LIN {X 0,Y 312.483,Z 213.378,A -85,B 0,C 180,E1 -15525.767,E2 -15525.767} C_VEL
LIN {X 0,Y 316.102,Z 224.16,A -85,B 0,C 180,E1 -15529.107,E2 -15529.107} C_VEL
LIN {X 0,Y 319.173,Z 234.249,A -85,B 0,C 180,E1 -15531.937,E2 -15531.937} C_VEL
LIN {X 0,Y 322.11,Z 245.048,A -85,B 0,C 180,E1 -15534.711,E2 -15534.711} C_VEL
LIN {X 0,Y 330.054,Z 261.785,A -85,B 0,C 180,E1 -15536.094,E2 -15536.094} C_VEL
LIN {X 0,Y 331.465,Z 265.176,A -85,B 0,C 180,E1 -15536.337,E2 -15536.337} C_VEL
LIN {X 0,Y 334.572,Z 286.176,A -85,B 0,C 180,E1 -15537.21,E2 -15537.21} C_VEL
LIN {X 0,Y 330.489,Z 404.791,A -85,B 0,C 180,E1 -15539.886,E2 -15539.886} C_VEL
LIN {X 0,Y 329.279,Z 420.508,A -85,B 0,C 180,E1 -15540.469,E2 -15540.469} C_VEL
LIN {X 0,Y 327.737,Z 434.949,A -85,B 0,C 180,E1 -15541.24,E2 -15541.24} C_VEL
LIN {X 0,Y 325.913,Z 449.505,A -85,B 0,C 180,E1 -15542.288,E2 -15542.288} C_VEL
LIN {X 0,Y 323.767,Z 463.536,A -85,B 0,C 180,E1 -15543.578,E2 -15543.578} C_VEL
LIN {X 0,Y 321.714,Z 475.702,A -85,B 0,C 180,E1 -15544.961,E2 -15544.961} C_VEL
LIN {X 0,Y 319.654,Z 487.038,A -85,B 0,C 180,E1 -15546.516,E2 -15546.516} C_VEL
LIN {X 0,Y 317.57,Z 498.142,A -85,B 0,C 180,E1 -15548.354,E2 -15548.354} C_VEL
LIN {X 0,Y 315.688,Z 508.785,A -85,B 0,C 180,E1 -15550.493,E2 -15550.493} C_VEL
LIN {X 0,Y 313.887,Z 518.044,A -85,B 0,C 180,E1 -15552.743,E2 -15552.743} C_VEL
LIN {X 0,Y 312.499,Z 526.423,A -85,B 0,C 180,E1 -15555.251,E2 -15555.251} C_VEL
LIN {X 0,Y 311.624,Z 532.842,A -85,B 0,C 180,E1 -15557.629,E2 -15557.629} C_VEL
LIN {X 0,Y 311.02,Z 538.401,A -85,B 0,C 180,E1 -15560.243,E2 -15560.243} C_VEL
LIN {X 0,Y 310.801,Z 541.607,A -85,B 0,C 180,E1 -15562.203,E2 -15562.203} C_VEL
LIN {X 0,Y 310.742,Z 544.767,A -85,B 0,C 180,E1 -15564.81,E2 -15564.81} C_VEL
LIN {X 0,Y 310.752,Z 546.649,A -85,B 0,C 180,E1 -15567.408,E2 -15567.408} C_VEL
LIN {X 0,Y 310.85,Z 547.287,A -85,B 0,C 180,E1 -15570,E2 -15570} C_VEL
LIN {X 0,Y 310.756,Z 546.639,A -85,B 0,C 180,E1 -15572.593,E2 -15572.593} C_VEL
LIN {X 0,Y 310.772,Z 544.746,A -85,B 0,C 180,E1 -15575.19,E2 -15575.19} C_VEL
LIN {X 0,Y 310.87,Z 541.581,A -85,B 0,C 180,E1 -15577.796,E2 -15577.796} C_VEL
LIN {X 0,Y 311.091,Z 537.073,A -85,B 0,C 180,E1 -15580.413,E2 -15580.413} C_VEL
LIN {X 0,Y 311.847,Z 531.123,A -85,B 0,C 180,E1 -15583.025,E2 -15583.025} C_VEL
LIN {X 0,Y 312.984,Z 523.568,A -85,B 0,C 180,E1 -15585.632,E2 -15585.632} C_VEL
LIN {X 0,Y 314.335,Z 515.443,A -85,B 0,C 180,E1 -15587.904,E2 -15587.904} C_VEL
LIN {X 0,Y 316.183,Z 505.652,A -85,B 0,C 180,E1 -15590.153,E2 -15590.153} C_VEL
LIN {X 0,Y 317.987,Z 495.61,A -85,B 0,C 180,E1 -15592.069,E2 -15592.069} C_VEL
LIN {X 0,Y 320.107,Z 483.635,A -85,B 0,C 180,E1 -15593.965,E2 -15593.965} C_VEL
LIN {X 0,Y 322.353,Z 471.672,A -85,B 0,C 180,E1 -15595.505,E2 -15595.505} C_VEL
LIN {X 0,Y 324.51,Z 458.681,A -85,B 0,C 180,E1 -15596.878,E2 -15596.878} C_VEL
LIN {X 0,Y 326.511,Z 444.201,A -85,B 0,C 180,E1 -15598.107,E2 -15598.107} C_VEL
LIN {X 0,Y 328.267,Z 429.502,A -85,B 0,C 180,E1 -15599.06,E2 -15599.06} C_VEL
LIN {X 0,Y 329.718,Z 414.75,A -85,B 0,C 180,E1 -15599.752,E2 -15599.752} C_VEL
LIN {X 0,Y 330.617,Z 399.638,A -85,B 0,C 180,E1 -15600.234,E2 -15600.234} C_VEL
LIN {X 0,Y 334.518,Z 285.951,A -85,B 0,C 180,E1 -15602.776,E2 -15602.776} C_VEL
LIN {X 0,Y 331.317,Z 264.741,A -85,B 0,C 180,E1 -15603.663,E2 -15603.663} C_VEL
LIN {X 0,Y 323.413,Z 247.872,A -85,B 0,C 180,E1 -15605.003,E2 -15605.003} C_VEL
LIN {X 0,Y 322.079,Z 244.847,A -85,B 0,C 180,E1 -15605.29,E2 -15605.29} C_VEL
LIN {X 0,Y 318.674,Z 232.493,A -85,B 0,C 180,E1 -15608.514,E2 -15608.514} C_VEL
LIN {X 0,Y 315.634,Z 222.757,A -85,B 0,C 180,E1 -15611.281,E2 -15611.281} C_VEL
LIN {X 0,Y 312.46,Z 213.28,A -85,B 0,C 180,E1 -15614.258,E2 -15614.258} C_VEL
LIN {X 0,Y 312.483,Z 213.169,A -85,B 0,C 180,E1 -15617.919,E2 -15617.919} C_VEL
LIN {X 0,Y 312.498,Z 213.176,A -85,B 0,C 180,E1 -15620.971,E2 -15620.971} C_VEL
LIN {X 0,Y 312.531,Z 213.179,A -85,B 0,C 180,E1 -15624.22,E2 -15624.22} C_VEL
LIN {X 0,Y 312.503,Z 213.157,A -85,B 0,C 180,E1 -15627.334,E2 -15627.334} C_VEL
LIN {X 0,Y 312.551,Z 213.17,A -85,B 0,C 180,E1 -15631.276,E2 -15631.276} C_VEL
LIN {X 0,Y 312.584,Z 213.149,A -85,B 0,C 180,E1 -15634.711,E2 -15634.711} C_VEL
LIN {X 0,Y 312.586,Z 213.171,A -85,B 0,C 180,E1 -15637.529,E2 -15637.529} C_VEL
LIN {X 0,Y 312.637,Z 213.16,A -85,B 0,C 180,E1 -15641.657,E2 -15641.657} C_VEL
LIN {X 0,Y 312.692,Z 213.152,A -85,B 0,C 180,E1 -15645.686,E2 -15645.686} C_VEL
LIN {X 0,Y 312.697,Z 213.151,A -85,B 0,C 180,E1 -15649.642,E2 -15649.642} C_VEL
LIN {X 0,Y 312.852,Z 213.141,A -85,B 0,C 180,E1 -15652.254,E2 -15652.254} C_VEL
LIN {X 0,Y 312.714,Z 213.146,A -85,B 0,C 180,E1 -15654.843,E2 -15654.843} C_VEL
LIN {X 0,Y 312.989,Z 213.111,A -85,B 0,C 180,E1 -15658.714,E2 -15658.714} C_VEL
LIN {X 0,Y 312.987,Z 213.124,A -85,B 0,C 180,E1 -15661.287,E2 -15661.287} C_VEL
LIN {X 0,Y 312.716,Z 213.156,A -85,B 0,C 180,E1 -15665.158,E2 -15665.158} C_VEL
LIN {X 0,Y 312.871,Z 213.127,A -85,B 0,C 180,E1 -15667.746,E2 -15667.746} C_VEL
LIN {X 0,Y 312.668,Z 213.152,A -85,B 0,C 180,E1 -15671.672,E2 -15671.672} C_VEL
LIN {X 0,Y 312.699,Z 213.155,A -85,B 0,C 180,E1 -15674.888,E2 -15674.888} C_VEL
LIN {X 0,Y 312.63,Z 213.16,A -85,B 0,C 180,E1 -15679.237,E2 -15679.237} C_VEL
LIN {X 0,Y 312.545,Z 213.174,A -85,B 0,C 180,E1 -15682.789,E2 -15682.789} C_VEL
LIN {X 0,Y 312.602,Z 213.17,A -85,B 0,C 180,E1 -15685.936,E2 -15685.936} C_VEL
LIN {X 0,Y 312.538,Z 213.151,A -85,B 0,C 180,E1 -15689.651,E2 -15689.651} C_VEL
LIN {X 0,Y 312.519,Z 213.162,A -85,B 0,C 180,E1 -15693.689,E2 -15693.689} C_VEL
LIN {X 0,Y 312.537,Z 213.18,A -85,B 0,C 180,E1 -15697.384,E2 -15697.384} C_VEL
LIN {X 0,Y 312.49,Z 213.168,A -85,B 0,C 180,E1 -15700.709,E2 -15700.709} C_VEL
LIN {X 0,Y 312.452,Z 213.173,A -85,B 0,C 180,E1 -15704.21,E2 -15704.21} C_VEL
LIN {X 0,Y 312.507,Z 213.373,A -85,B 0,C 180,E1 -15708.078,E2 -15708.078} C_VEL
LIN {X 0,Y 315.863,Z 224.153,A -85,B 0,C 180,E1 -15711.657,E2 -15711.657} C_VEL
LIN {X 0,Y 319.038,Z 235.379,A -85,B 0,C 180,E1 -15715.058,E2 -15715.058} C_VEL
LIN {X 0,Y 321.292,Z 244.626,A -85,B 0,C 180,E1 -15717.605,E2 -15717.605} C_VEL
LIN {X 0,Y 328.843,Z 260.881,A -85,B 0,C 180,E1 -15718.909,E2 -15718.909} C_VEL
LIN {X 0,Y 333.903,Z 287.047,A -85,B 0,C 180,E1 -15720.083,E2 -15720.083} C_VEL
LIN {X 0,Y 331.092,Z 389.615,A -85,B 0,C 180,E1 -15722.204,E2 -15722.204} C_VEL
LIN {X 0,Y 330.174,Z 403.917,A -85,B 0,C 180,E1 -15722.722,E2 -15722.722} C_VEL
LIN {X 0,Y 329.016,Z 417.284,A -85,B 0,C 180,E1 -15723.442,E2 -15723.442} C_VEL
LIN {X 0,Y 327.379,Z 430.378,A -85,B 0,C 180,E1 -15724.374,E2 -15724.374} C_VEL
LIN {X 0,Y 325.773,Z 442.564,A -85,B 0,C 180,E1 -15725.504,E2 -15725.504} C_VEL
LIN {X 0,Y 323.801,Z 454.245,A -85,B 0,C 180,E1 -15726.834,E2 -15726.834} C_VEL
LIN {X 0,Y 321.813,Z 464.206,A -85,B 0,C 180,E1 -15728.207,E2 -15728.207} C_VEL
LIN {X 0,Y 320.008,Z 473.526,A -85,B 0,C 180,E1 -15729.763,E2 -15729.763} C_VEL
LIN {X 0,Y 317.924,Z 482.935,A -85,B 0,C 180,E1 -15731.638,E2 -15731.638} C_VEL
LIN {X 0,Y 316.379,Z 490.759,A -85,B 0,C 180,E1 -15733.547,E2 -15733.547} C_VEL
LIN {X 0,Y 314.546,Z 498.315,A -85,B 0,C 180,E1 -15735.772,E2 -15735.772} C_VEL
LIN {X 0,Y 313.128,Z 505.191,A -85,B 0,C 180,E1 -15738.346,E2 -15738.346} C_VEL
LIN {X 0,Y 312.133,Z 510.443,A -85,B 0,C 180,E1 -15740.931,E2 -15740.931} C_VEL
LIN {X 0,Y 311.505,Z 514.238,A -85,B 0,C 180,E1 -15743.522,E2 -15743.522} C_VEL
LIN {X 0,Y 311.057,Z 516.717,A -85,B 0,C 180,E1 -15746.113,E2 -15746.113} C_VEL
LIN {X 0,Y 310.876,Z 517.952,A -85,B 0,C 180,E1 -15748.704,E2 -15748.704} C_VEL
LIN {X 0,Y 310.869,Z 517.977,A -85,B 0,C 180,E1 -15751.295,E2 -15751.295} C_VEL
LIN {X 0,Y 311.046,Z 516.796,A -85,B 0,C 180,E1 -15753.886,E2 -15753.886} C_VEL
LIN {X 0,Y 311.478,Z 514.372,A -85,B 0,C 180,E1 -15756.477,E2 -15756.477} C_VEL
LIN {X 0,Y 312.074,Z 510.638,A -85,B 0,C 180,E1 -15759.069,E2 -15759.069} C_VEL
LIN {X 0,Y 313.084,Z 505.458,A -85,B 0,C 180,E1 -15761.655,E2 -15761.655} C_VEL
LIN {X 0,Y 314.484,Z 498.657,A -85,B 0,C 180,E1 -15764.23,E2 -15764.23} C_VEL
LIN {X 0,Y 316.288,Z 491.172,A -85,B 0,C 180,E1 -15766.457,E2 -15766.457} C_VEL
LIN {X 0,Y 317.855,Z 483.429,A -85,B 0,C 180,E1 -15768.365,E2 -15768.365} C_VEL
LIN {X 0,Y 319.886,Z 474.122,A -85,B 0,C 180,E1 -15770.244,E2 -15770.244} C_VEL
LIN {X 0,Y 321.942,Z 463.859,A -85,B 0,C 180,E1 -15771.952,E2 -15771.952} C_VEL
LIN {X 0,Y 324.092,Z 452.583,A -85,B 0,C 180,E1 -15773.481,E2 -15773.481} C_VEL
LIN {X 0,Y 326.143,Z 440.017,A -85,B 0,C 180,E1 -15774.861,E2 -15774.861} C_VEL
LIN {X 0,Y 327.889,Z 427.288,A -85,B 0,C 180,E1 -15775.97,E2 -15775.97} C_VEL
LIN {X 0,Y 329.37,Z 413.766,A -85,B 0,C 180,E1 -15776.877,E2 -15776.877} C_VEL
LIN {X 0,Y 330.53,Z 400.017,A -85,B 0,C 180,E1 -15777.545,E2 -15777.545} C_VEL
LIN {X 0,Y 331.251,Z 386.055,A -85,B 0,C 180,E1 -15777.995,E2 -15777.995} C_VEL
LIN {X 0,Y 333.983,Z 287.076,A -85,B 0,C 180,E1 -15780.023,E2 -15780.023} C_VEL
LIN {X 0,Y 332.453,Z 278.562,A -85,B 0,C 180,E1 -15780.386,E2 -15780.386} C_VEL
LIN {X 0,Y 330.934,Z 273.085,A -85,B 0,C 180,E1 -15780.681,E2 -15780.681} C_VEL
LIN {X 0,Y 328.544,Z 268.082,A -85,B 0,C 180,E1 -15781.065,E2 -15781.065} C_VEL
LIN {X 0,Y 322.423,Z 259.006,A -85,B 0,C 180,E1 -15781.989,E2 -15781.989} C_VEL
LIN {X 0,Y 318.247,Z 253.023,A -85,B 0,C 180,E1 -15782.64,E2 -15782.64} C_VEL
LIN {X 0,Y 314.109,Z 244.538,A -85,B 0,C 180,E1 -15783.413,E2 -15783.413} C_VEL
LIN {X 0,Y 311.656,Z 234.748,A -85,B 0,C 180,E1 -15786.246,E2 -15786.246} C_VEL
LIN {X 0,Y 308.577,Z 224.118,A -85,B 0,C 180,E1 -15789.62,E2 -15789.62} C_VEL
LIN {X 0,Y 305.432,Z 214.127,A -85,B 0,C 180,E1 -15793.142,E2 -15793.142} C_VEL
LIN {X 0,Y 305.452,Z 214.059,A -85,B 0,C 180,E1 -15797.413,E2 -15797.413} C_VEL
LIN {X 0,Y 305.491,Z 214.047,A -85,B 0,C 180,E1 -15801.599,E2 -15801.599} C_VEL
LIN {X 0,Y 305.458,Z 214.036,A -85,B 0,C 180,E1 -15804.886,E2 -15804.886} C_VEL
LIN {X 0,Y 305.449,Z 214.063,A -85,B 0,C 180,E1 -15808.354,E2 -15808.354} C_VEL
LIN {X 0,Y 305.516,Z 214.02,A -85,B 0,C 180,E1 -15811.113,E2 -15811.113} C_VEL
LIN {X 0,Y 305.567,Z 214.046,A -85,B 0,C 180,E1 -15814.087,E2 -15814.087} C_VEL
LIN {X 0,Y 305.522,Z 214.053,A -85,B 0,C 180,E1 -15818.404,E2 -15818.404} C_VEL
LIN {X 0,Y 305.585,Z 214.041,A -85,B 0,C 180,E1 -15821.217,E2 -15821.217} C_VEL
LIN {X 0,Y 305.643,Z 214.036,A -85,B 0,C 180,E1 -15825.348,E2 -15825.348} C_VEL
LIN {X 0,Y 305.632,Z 214.037,A -85,B 0,C 180,E1 -15829.399,E2 -15829.399} C_VEL
LIN {X 0,Y 305.807,Z 214.008,A -85,B 0,C 180,E1 -15832.074,E2 -15832.074} C_VEL
LIN {X 0,Y 305.683,Z 214.034,A -85,B 0,C 180,E1 -15834.723,E2 -15834.723} C_VEL
LIN {X 0,Y 305.951,Z 214.001,A -85,B 0,C 180,E1 -15838.684,E2 -15838.684} C_VEL
LIN {X 0,Y 305.951,Z 213.987,A -85,B 0,C 180,E1 -15841.316,E2 -15841.316} C_VEL
LIN {X 0,Y 305.846,Z 214.007,A -85,B 0,C 180,E1 -15846.597,E2 -15846.597} C_VEL
LIN {X 0,Y 305.73,Z 214.018,A -85,B 0,C 180,E1 -15849.26,E2 -15849.26} C_VEL
LIN {X 0,Y 305.582,Z 214.037,A -85,B 0,C 180,E1 -15853.296,E2 -15853.296} C_VEL
LIN {X 0,Y 305.587,Z 214.045,A -85,B 0,C 180,E1 -15856.02,E2 -15856.02} C_VEL
LIN {X 0,Y 305.571,Z 214.046,A -85,B 0,C 180,E1 -15859.445,E2 -15859.445} C_VEL
LIN {X 0,Y 305.485,Z 214.057,A -85,B 0,C 180,E1 -15863.042,E2 -15863.042} C_VEL
LIN {X 0,Y 305.52,Z 214.019,A -85,B 0,C 180,E1 -15866.219,E2 -15866.219} C_VEL
LIN {X 0,Y 305.49,Z 214.055,A -85,B 0,C 180,E1 -15869.05,E2 -15869.05} C_VEL
LIN {X 0,Y 305.459,Z 214.038,A -85,B 0,C 180,E1 -15873.517,E2 -15873.517} C_VEL
LIN {X 0,Y 305.467,Z 214.043,A -85,B 0,C 180,E1 -15876.74,E2 -15876.74} C_VEL
LIN {X 0,Y 305.449,Z 214.055,A -85,B 0,C 180,E1 -15880.6,E2 -15880.6} C_VEL
LIN {X 0,Y 305.42,Z 214.065,A -85,B 0,C 180,E1 -15883.656,E2 -15883.656} C_VEL
LIN {X 0,Y 305.451,Z 214.348,A -85,B 0,C 180,E1 -15884.793,E2 -15884.793} C_VEL
LIN {X 0,Y 309.409,Z 226.078,A -85,B 0,C 180,E1 -15888.553,E2 -15888.553} C_VEL
LIN {X 0,Y 312.373,Z 235.741,A -85,B 0,C 180,E1 -15891.363,E2 -15891.363} C_VEL
LIN {X 0,Y 314.93,Z 245.01,A -85,B 0,C 180,E1 -15893.826,E2 -15893.826} C_VEL
LIN {X 0,Y 323.133,Z 261.948,A -85,B 0,C 180,E1 -15895.314,E2 -15895.314} C_VEL
LIN {X 0,Y 325.651,Z 267.579,A -85,B 0,C 180,E1 -15895.754,E2 -15895.754} C_VEL
LIN {X 0,Y 328.503,Z 287.414,A -85,B 0,C 180,E1 -15896.595,E2 -15896.595} C_VEL
LIN {X 0,Y 324.346,Z 403.742,A -85,B 0,C 180,E1 -15899.255,E2 -15899.255} C_VEL
LIN {X 0,Y 323.177,Z 419.01,A -85,B 0,C 180,E1 -15899.81,E2 -15899.81} C_VEL
LIN {X 0,Y 321.508,Z 434.4,A -85,B 0,C 180,E1 -15900.629,E2 -15900.629} C_VEL
LIN {X 0,Y 319.548,Z 449.023,A -85,B 0,C 180,E1 -15901.687,E2 -15901.687} C_VEL
LIN {X 0,Y 317.388,Z 463.102,A -85,B 0,C 180,E1 -15903.004,E2 -15903.004} C_VEL
LIN {X 0,Y 315.22,Z 475.296,A -85,B 0,C 180,E1 -15904.408,E2 -15904.408} C_VEL
LIN {X 0,Y 313.057,Z 486.644,A -85,B 0,C 180,E1 -15905.991,E2 -15905.991} C_VEL
LIN {X 0,Y 310.734,Z 498.593,A -85,B 0,C 180,E1 -15908.02,E2 -15908.02} C_VEL
LIN {X 0,Y 308.92,Z 508.423,A -85,B 0,C 180,E1 -15910.048,E2 -15910.048} C_VEL
LIN {X 0,Y 307.051,Z 517.693,A -85,B 0,C 180,E1 -15912.346,E2 -15912.346} C_VEL
LIN {X 0,Y 305.681,Z 525.37,A -85,B 0,C 180,E1 -15914.67,E2 -15914.67} C_VEL
LIN {X 0,Y 304.617,Z 532.499,A -85,B 0,C 180,E1 -15917.34,E2 -15917.34} C_VEL
LIN {X 0,Y 303.947,Z 538.061,A -85,B 0,C 180,E1 -15920.014,E2 -15920.014} C_VEL
LIN {X 0,Y 303.741,Z 541.272,A -85,B 0,C 180,E1 -15922.021,E2 -15922.021} C_VEL
LIN {X 0,Y 303.684,Z 544.435,A -85,B 0,C 180,E1 -15924.689,E2 -15924.689} C_VEL
LIN {X 0,Y 303.672,Z 546.317,A -85,B 0,C 180,E1 -15927.348,E2 -15927.348} C_VEL
LIN {X 0,Y 303.757,Z 546.954,A -85,B 0,C 180,E1 -15930,E2 -15930} C_VEL
LIN {X 0,Y 303.678,Z 546.307,A -85,B 0,C 180,E1 -15932.653,E2 -15932.653} C_VEL
LIN {X 0,Y 303.685,Z 544.411,A -85,B 0,C 180,E1 -15935.312,E2 -15935.312} C_VEL
LIN {X 0,Y 303.79,Z 541.243,A -85,B 0,C 180,E1 -15937.979,E2 -15937.979} C_VEL
LIN {X 0,Y 304.043,Z 536.731,A -85,B 0,C 180,E1 -15940.657,E2 -15940.657} C_VEL
LIN {X 0,Y 304.852,Z 530.778,A -85,B 0,C 180,E1 -15943.329,E2 -15943.329} C_VEL
